Yaskawa INFORM job: DEMO_ROOF_SIDE_0625_3PAINT_18.JBI

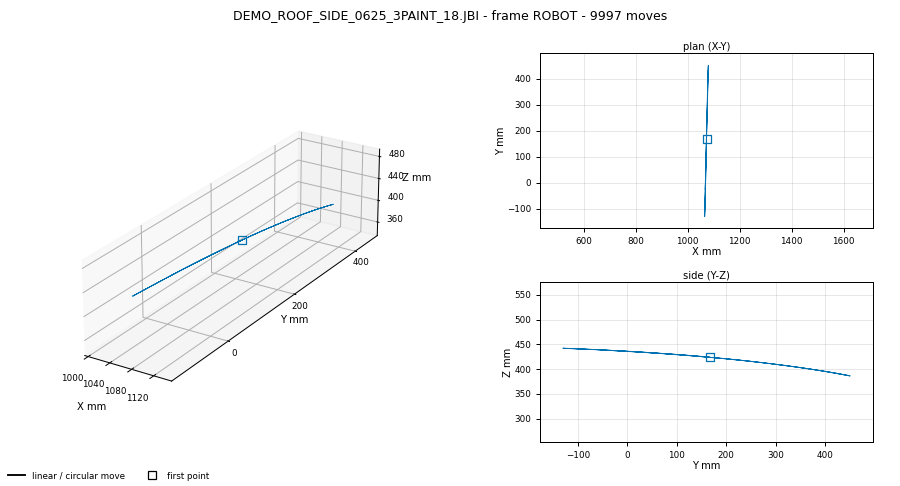
[picture p0: tool path of DEMO_ROOF_SIDE_0625_3PAINT_18.JBI in frame ROBOT, 9997 of 9997 moves have a stored position in this frame; points joined in program order, loops and branches not executed]
/JOB
//NAME DEMO_ROOF_SIDE_0625_3PAINT18
//POS
///NPOS 9997,0,0,0,0,0
///TOOL 0
///USER 0
///POSTYPE ROBOT
///RECTAN
///RCONF 1,0,0,0,0,0,0,0,0,0,0,0,0,0,0,0,0,0,0,0,0,0,0,0
C00000=1073.553,166.231,424.191,173.717,26.118,154.637
C00001=1073.548,165.982,424.213,173.714,26.115,154.636
C00002=1073.541,165.733,424.236,173.713,26.113,154.636
C00003=1073.536,165.484,424.258,173.710,26.110,154.636
C00004=1073.531,165.235,424.280,173.709,26.108,154.635
C00005=1073.525,164.986,424.301,173.707,26.105,154.635
C00006=1073.520,164.737,424.323,173.705,26.102,154.635
C00007=1073.514,164.488,424.345,173.703,26.099,154.634
C00008=1073.509,164.239,424.367,173.701,26.097,154.634
C00009=1073.503,163.990,424.389,173.699,26.094,154.634
C00010=1073.498,163.742,424.411,173.697,26.092,154.633
C00011=1073.492,163.492,424.433,173.695,26.088,154.633
C00012=1073.487,163.244,424.454,173.694,26.086,154.633
C00013=1073.481,162.994,424.477,173.691,26.083,154.632
C00014=1073.476,162.746,424.498,173.690,26.081,154.632
C00015=1073.470,162.496,424.520,173.688,26.078,154.632
C00016=1073.465,162.248,424.541,173.685,26.075,154.631
C00017=1073.459,161.998,424.564,173.684,26.072,154.631
C00018=1073.454,161.750,424.585,173.681,26.069,154.631
C00019=1073.448,161.500,424.607,173.680,26.067,154.630
C00020=1073.443,161.252,424.628,173.678,26.064,154.630
C00021=1073.437,161.002,424.650,173.676,26.061,154.630
C00022=1073.432,160.754,424.672,173.674,26.059,154.629
C00023=1073.426,160.504,424.694,173.672,26.056,154.629
C00024=1073.420,160.255,424.715,173.670,26.054,154.629
C00025=1073.414,160.007,424.736,173.669,26.051,154.628
C00026=1073.409,159.757,424.759,173.666,26.048,154.628
C00027=1073.402,159.475,424.782,173.665,26.045,154.628
C00028=1073.396,159.194,424.807,173.662,26.042,154.627
C00029=1073.390,158.911,424.831,173.660,26.040,154.627
C00030=1073.383,158.630,424.856,173.658,26.036,154.627
C00031=1073.377,158.381,424.877,173.656,26.034,154.626
C00032=1073.372,158.132,424.898,173.654,26.031,154.626
C00033=1073.366,157.882,424.920,173.653,26.028,154.625
C00034=1073.360,157.634,424.941,173.650,26.026,154.625
C00035=1073.355,157.384,424.963,173.649,26.023,154.625
C00036=1073.349,157.136,424.984,173.646,26.020,154.625
C00037=1073.343,156.887,425.006,173.645,26.018,154.624
C00038=1073.338,156.638,425.027,173.643,26.015,154.624
C00039=1073.332,156.388,425.048,173.641,26.013,154.624
C00040=1073.326,156.140,425.070,173.639,26.010,154.623
C00041=1073.321,155.890,425.092,173.637,26.007,154.623
C00042=1073.315,155.641,425.112,173.635,26.005,154.623
C00043=1073.310,155.393,425.134,173.634,26.002,154.622
C00044=1073.304,155.144,425.155,173.631,25.999,154.622
C00045=1073.298,154.895,425.176,173.630,25.997,154.622
C00046=1073.292,154.645,425.197,173.627,25.994,154.621
C00047=1073.287,154.397,425.219,173.626,25.992,154.621
C00048=1073.281,154.147,425.240,173.624,25.989,154.621
C00049=1073.275,153.899,425.262,173.622,25.986,154.620
C00050=1073.269,153.649,425.282,173.621,25.984,154.620
C00051=1073.264,153.401,425.304,173.618,25.981,154.620
C00052=1073.258,153.151,425.326,173.617,25.978,154.619
C00053=1073.253,152.902,425.347,173.614,25.975,154.619
C00054=1073.247,152.654,425.368,173.613,25.973,154.619
C00055=1073.241,152.404,425.389,173.611,25.970,154.618
C00056=1073.236,152.155,425.410,173.609,25.968,154.618
C00057=1073.230,151.906,425.432,173.607,25.965,154.618
C00058=1073.225,151.657,425.452,173.605,25.962,154.617
C00059=1073.219,151.408,425.473,173.604,25.960,154.617
C00060=1073.213,151.159,425.494,173.602,25.957,154.617
C00061=1073.208,150.910,425.516,173.600,25.955,154.616
C00062=1073.201,150.661,425.537,173.598,25.952,154.616
C00063=1073.196,150.412,425.558,173.596,25.949,154.616
C00064=1073.191,150.163,425.579,173.594,25.947,154.615
C00065=1073.185,149.913,425.600,173.593,25.944,154.615
C00066=1073.179,149.665,425.621,173.590,25.941,154.615
C00067=1073.174,149.416,425.642,173.589,25.939,154.615
C00068=1073.168,149.167,425.663,173.587,25.936,154.614
C00069=1073.162,148.917,425.684,173.585,25.933,154.614
C00070=1073.156,148.668,425.706,173.584,25.931,154.613
C00071=1073.150,148.419,425.726,173.581,25.928,154.613
C00072=1073.145,148.171,425.747,173.580,25.925,154.613
C00073=1073.139,147.921,425.768,173.577,25.923,154.613
C00074=1073.133,147.673,425.789,173.576,25.920,154.612
C00075=1073.128,147.423,425.810,173.575,25.918,154.612
C00076=1073.122,147.174,425.831,173.572,25.915,154.612
C00077=1073.117,146.925,425.852,173.571,25.913,154.611
C00078=1073.111,146.676,425.872,173.568,25.909,154.611
C00079=1073.104,146.427,425.893,173.567,25.907,154.611
C00080=1073.099,146.178,425.914,173.565,25.905,154.610
C00081=1073.094,145.929,425.935,173.563,25.902,154.610
C00082=1073.088,145.680,425.956,173.562,25.900,154.610
C00083=1073.082,145.431,425.976,173.559,25.896,154.609
C00084=1073.076,145.182,425.997,173.558,25.894,154.609
C00085=1073.070,144.932,426.018,173.555,25.891,154.609
C00086=1073.065,144.683,426.039,173.554,25.889,154.608
C00087=1073.060,144.435,426.060,173.553,25.886,154.608
C00088=1073.053,144.185,426.080,173.550,25.883,154.608
C00089=1073.048,143.936,426.101,173.549,25.881,154.607
C00090=1073.042,143.687,426.122,173.546,25.878,154.607
C00091=1073.036,143.405,426.145,173.545,25.876,154.607
C00092=1073.029,143.123,426.169,173.543,25.872,154.606
C00093=1073.023,142.841,426.193,173.540,25.869,154.606
C00094=1073.017,142.559,426.215,173.539,25.866,154.606
C00095=1073.011,142.310,426.237,173.537,25.864,154.605
C00096=1073.005,142.060,426.258,173.535,25.861,154.605
C00097=1072.999,141.812,426.278,173.533,25.858,154.605
C00098=1072.994,141.562,426.298,173.532,25.856,154.604
C00099=1072.989,141.313,426.319,173.530,25.853,154.604
C00100=1072.983,141.064,426.340,173.528,25.850,154.604
C00101=1072.977,140.815,426.360,173.526,25.848,154.603
C00102=1072.971,140.566,426.381,173.525,25.845,154.603
C00103=1072.966,140.317,426.401,173.523,25.842,154.603
C00104=1072.959,140.068,426.422,173.521,25.840,154.602
C00105=1072.954,139.818,426.442,173.519,25.837,154.602
C00106=1072.949,139.570,426.463,173.517,25.835,154.602
C00107=1072.943,139.321,426.483,173.516,25.832,154.601
C00108=1072.937,139.071,426.504,173.514,25.829,154.601
C00109=1072.931,138.822,426.524,173.512,25.827,154.601
C00110=1072.926,138.573,426.545,173.511,25.824,154.600
C00111=1072.920,138.324,426.565,173.508,25.822,154.600
C00112=1072.914,138.075,426.585,173.507,25.819,154.600
C00113=1072.908,137.826,426.606,173.505,25.816,154.599
C00114=1072.902,137.577,426.626,173.503,25.814,154.599
C00115=1072.897,137.328,426.647,173.502,25.811,154.599
C00116=1072.891,137.079,426.667,173.499,25.808,154.598
C00117=1072.886,136.830,426.687,173.498,25.806,154.598
C00118=1072.880,136.580,426.708,173.497,25.803,154.598
C00119=1072.874,136.332,426.729,173.494,25.801,154.597
C00120=1072.869,136.083,426.749,173.493,25.798,154.597
C00121=1072.863,135.834,426.769,173.491,25.796,154.597
C00122=1072.858,135.584,426.789,173.489,25.792,154.596
C00123=1072.851,135.334,426.810,173.488,25.790,154.596
C00124=1072.846,135.085,426.830,173.485,25.788,154.596
C00125=1072.840,134.837,426.850,173.484,25.785,154.595
C00126=1072.834,134.587,426.871,173.482,25.782,154.595
C00127=1072.828,134.339,426.891,173.480,25.779,154.595
C00128=1072.823,134.089,426.911,173.479,25.777,154.594
C00129=1072.817,133.841,426.931,173.477,25.774,154.594
C00130=1072.811,133.591,426.952,173.475,25.772,154.594
C00131=1072.805,133.342,426.972,173.473,25.769,154.593
C00132=1072.800,133.093,426.993,173.472,25.766,154.593
C00133=1072.794,132.844,427.013,173.470,25.764,154.593
C00134=1072.789,132.595,427.033,173.468,25.761,154.592
C00135=1072.783,132.346,427.052,173.467,25.759,154.592
C00136=1072.778,132.096,427.073,173.465,25.755,154.592
C00137=1072.772,131.848,427.093,173.463,25.753,154.591
C00138=1072.765,131.598,427.113,173.462,25.750,154.591
C00139=1072.760,131.349,427.134,173.459,25.748,154.591
C00140=1072.754,131.100,427.154,173.458,25.745,154.591
C00141=1072.748,130.851,427.173,173.456,25.743,154.590
C00142=1072.742,130.602,427.193,173.454,25.740,154.590
C00143=1072.737,130.353,427.213,173.453,25.738,154.590
C00144=1072.731,130.103,427.234,173.451,25.735,154.589
C00145=1072.725,129.854,427.254,173.449,25.732,154.589
C00146=1072.719,129.605,427.273,173.447,25.730,154.589
C00147=1072.714,129.356,427.294,173.446,25.727,154.588
C00148=1072.708,129.107,427.313,173.444,25.725,154.588
C00149=1072.702,128.858,427.333,173.442,25.722,154.588
C00150=1072.696,128.609,427.353,173.441,25.719,154.587
C00151=1072.691,128.360,427.373,173.438,25.717,154.587
C00152=1072.684,128.110,427.394,173.437,25.714,154.587
C00153=1072.678,127.861,427.413,173.436,25.712,154.586
C00154=1072.672,127.612,427.433,173.434,25.709,154.586
C00155=1072.666,127.330,427.455,173.432,25.706,154.586
C00156=1072.660,127.047,427.478,173.430,25.703,154.585
C00157=1072.653,126.765,427.500,173.428,25.700,154.585
C00158=1072.647,126.483,427.523,173.426,25.697,154.584
C00159=1072.641,126.234,427.543,173.425,25.695,154.584
C00160=1072.635,125.985,427.562,173.422,25.692,154.584
C00161=1072.630,125.736,427.583,173.421,25.689,154.584
C00162=1072.624,125.487,427.603,173.419,25.687,154.583
C00163=1072.618,125.237,427.622,173.418,25.684,154.583
C00164=1072.612,124.989,427.642,173.416,25.682,154.583
C00165=1072.606,124.739,427.661,173.414,25.679,154.582
C00166=1072.600,124.490,427.681,173.413,25.676,154.582
C00167=1072.595,124.241,427.702,173.410,25.674,154.582
C00168=1072.589,123.992,427.721,173.409,25.671,154.581
C00169=1072.583,123.743,427.741,173.408,25.669,154.581
C00170=1072.578,123.494,427.760,173.405,25.665,154.581
C00171=1072.572,123.245,427.780,173.404,25.663,154.580
C00172=1072.566,122.995,427.799,173.403,25.660,154.580
C00173=1072.561,122.746,427.820,173.401,25.658,154.580
C00174=1072.555,122.497,427.839,173.399,25.655,154.579
C00175=1072.549,122.248,427.859,173.397,25.653,154.579
C00176=1072.543,121.998,427.878,173.396,25.650,154.578
C00177=1072.537,121.750,427.898,173.394,25.647,154.578
C00178=1072.532,121.500,427.917,173.392,25.644,154.578
C00179=1072.526,121.251,427.938,173.391,25.642,154.578
C00180=1072.521,121.002,427.957,173.389,25.640,154.577
C00181=1072.515,120.753,427.977,173.387,25.637,154.577
C00182=1072.509,120.503,427.996,173.386,25.634,154.577
C00183=1072.503,120.254,428.016,173.384,25.631,154.576
C00184=1072.497,120.005,428.036,173.383,25.629,154.576
C00185=1072.492,119.756,428.055,173.381,25.626,154.576
C00186=1072.486,119.507,428.075,173.379,25.624,154.575
C00187=1072.481,119.257,428.095,173.378,25.621,154.575
C00188=1072.475,119.008,428.114,173.375,25.618,154.575
C00189=1072.469,118.759,428.134,173.374,25.615,154.574
C00190=1072.464,118.510,428.153,173.373,25.612,154.574
C00191=1072.458,118.261,428.173,173.371,25.610,154.573
C00192=1072.452,118.012,428.192,173.369,25.607,154.573
C00193=1072.447,117.763,428.211,173.368,25.605,154.573
C00194=1072.441,117.514,428.231,173.366,25.602,154.572
C00195=1072.435,117.264,428.250,173.365,25.600,154.572
C00196=1072.430,117.015,428.270,173.362,25.596,154.572
C00197=1072.424,116.765,428.289,173.361,25.594,154.571
C00198=1072.419,116.517,428.309,173.360,25.591,154.571
C00199=1072.413,116.268,428.328,173.358,25.589,154.571
C00200=1072.408,116.018,428.348,173.356,25.586,154.570
C00201=1072.402,115.769,428.367,173.355,25.583,154.570
C00202=1072.396,115.520,428.387,173.353,25.581,154.570
C00203=1072.390,115.270,428.406,173.352,25.578,154.569
C00204=1072.385,115.022,428.425,173.349,25.575,154.569
C00205=1072.379,114.773,428.445,173.348,25.572,154.569
C00206=1072.373,114.523,428.464,173.347,25.570,154.568
C00207=1072.368,114.274,428.483,173.345,25.567,154.568
C00208=1072.362,114.025,428.503,173.343,25.564,154.568
C00209=1072.356,113.775,428.522,173.342,25.562,154.567
C00210=1072.350,113.526,428.542,173.340,25.559,154.567
C00211=1072.345,113.278,428.561,173.339,25.556,154.567
C00212=1072.340,113.028,428.580,173.336,25.554,154.566
C00213=1072.334,112.779,428.599,173.335,25.551,154.566
C00214=1072.328,112.530,428.618,173.334,25.549,154.566
C00215=1072.322,112.280,428.637,173.332,25.546,154.565
C00216=1072.316,112.031,428.656,173.330,25.543,154.565
C00217=1072.310,111.782,428.676,173.329,25.540,154.565
C00218=1072.305,111.533,428.695,173.327,25.538,154.564
C00219=1072.298,111.251,428.716,173.325,25.535,154.564
C00220=1072.292,110.968,428.738,173.324,25.532,154.563
C00221=1072.285,110.686,428.760,173.321,25.529,154.563
C00222=1072.278,110.403,428.781,173.320,25.526,154.563
C00223=1072.273,110.155,428.800,173.318,25.523,154.562
C00224=1072.267,109.905,428.819,173.316,25.520,154.562
C00225=1072.262,109.656,428.839,173.315,25.518,154.562
C00226=1072.255,109.407,428.857,173.314,25.515,154.561
C00227=1072.249,109.157,428.876,173.312,25.513,154.561
C00228=1072.244,108.908,428.896,173.310,25.510,154.561
C00229=1072.239,108.659,428.915,173.308,25.507,154.560
C00230=1072.232,108.410,428.933,173.307,25.505,154.560
C00231=1072.227,108.160,428.953,173.306,25.502,154.560
C00232=1072.221,107.911,428.972,173.303,25.500,154.559
C00233=1072.214,107.662,428.990,173.302,25.497,154.559
C00234=1072.209,107.413,429.009,173.300,25.495,154.559
C00235=1072.204,107.164,429.029,173.299,25.492,154.558
C00236=1072.197,106.915,429.047,173.298,25.489,154.558
C00237=1072.192,106.665,429.066,173.295,25.486,154.558
C00238=1072.186,106.416,429.086,173.294,25.484,154.557
C00239=1072.181,106.167,429.105,173.293,25.481,154.557
C00240=1072.174,105.918,429.123,173.291,25.479,154.557
C00241=1072.169,105.669,429.142,173.289,25.476,154.556
C00242=1072.163,105.419,429.162,173.288,25.473,154.556
C00243=1072.157,105.171,429.180,173.286,25.470,154.556
C00244=1072.152,104.921,429.198,173.285,25.468,154.555
C00245=1072.146,104.671,429.218,173.283,25.465,154.555
C00246=1072.140,104.423,429.236,173.281,25.463,154.555
C00247=1072.135,104.173,429.255,173.280,25.460,154.554
C00248=1072.129,103.924,429.274,173.278,25.457,154.554
C00249=1072.122,103.675,429.293,173.277,25.455,154.554
C00250=1072.117,103.426,429.312,173.276,25.452,154.553
C00251=1072.112,103.176,429.331,173.273,25.449,154.553
C00252=1072.106,102.927,429.349,173.272,25.446,154.553
C00253=1072.100,102.678,429.368,173.271,25.444,154.552
C00254=1072.094,102.429,429.387,173.269,25.441,154.552
C00255=1072.088,102.180,429.406,173.268,25.439,154.552
C00256=1072.084,101.930,429.424,173.266,25.435,154.551
C00257=1072.077,101.681,429.443,173.264,25.433,154.551
C00258=1072.071,101.432,429.462,173.263,25.430,154.550
C00259=1072.066,101.183,429.481,173.261,25.427,154.550
C00260=1072.060,100.933,429.499,173.260,25.425,154.550
C00261=1072.055,100.684,429.518,173.258,25.422,154.550
C00262=1072.048,100.435,429.537,173.256,25.420,154.549
C00263=1072.042,100.186,429.555,173.255,25.417,154.549
C00264=1072.037,99.936,429.574,173.254,25.414,154.548
C00265=1072.030,99.687,429.592,173.252,25.412,154.548
C00266=1072.025,99.438,429.611,173.250,25.409,154.548
C00267=1072.019,99.189,429.629,173.248,25.407,154.547
C00268=1072.014,98.939,429.648,173.247,25.404,154.547
C00269=1072.007,98.690,429.667,173.246,25.401,154.547
C00270=1072.002,98.441,429.684,173.244,25.399,154.546
C00271=1071.996,98.192,429.704,173.242,25.396,154.546
C00272=1071.990,97.942,429.722,173.241,25.393,154.546
C00273=1071.985,97.693,429.740,173.239,25.391,154.545
C00274=1071.978,97.444,429.759,173.238,25.388,154.545
C00275=1071.973,97.194,429.778,173.236,25.386,154.545
C00276=1071.967,96.945,429.796,173.234,25.382,154.544
C00277=1071.961,96.696,429.815,173.233,25.380,154.544
C00278=1071.956,96.447,429.833,173.231,25.377,154.544
C00279=1071.949,96.198,429.851,173.230,25.375,154.543
C00280=1071.944,95.948,429.870,173.229,25.372,154.543
C00281=1071.938,95.699,429.888,173.227,25.370,154.543
C00282=1071.932,95.450,429.906,173.225,25.367,154.542
C00283=1071.926,95.168,429.927,173.224,25.364,154.542
C00284=1071.919,94.885,429.949,173.221,25.360,154.542
C00285=1071.913,94.604,429.969,173.220,25.358,154.541
C00286=1071.906,94.321,429.990,173.219,25.355,154.541
C00287=1071.900,94.072,430.008,173.217,25.352,154.540
C00288=1071.895,93.822,430.027,173.215,25.349,154.540
C00289=1071.889,93.573,430.045,173.214,25.346,154.540
C00290=1071.883,93.324,430.064,173.212,25.344,154.539
C00291=1071.877,93.074,430.082,173.211,25.341,154.539
C00292=1071.871,92.826,430.100,173.209,25.338,154.539
C00293=1071.866,92.576,430.119,173.207,25.336,154.538
C00294=1071.861,92.327,430.136,173.206,25.333,154.538
C00295=1071.854,92.078,430.155,173.205,25.330,154.538
C00296=1071.849,91.828,430.173,173.203,25.328,154.537
C00297=1071.843,91.579,430.192,173.202,25.325,154.537
C00298=1071.837,91.329,430.210,173.200,25.322,154.537
C00299=1071.832,91.081,430.228,173.198,25.320,154.536
C00300=1071.826,90.831,430.246,173.197,25.317,154.536
C00301=1071.820,90.582,430.264,173.196,25.315,154.536
C00302=1071.814,90.333,430.283,173.194,25.312,154.535
C00303=1071.808,90.084,430.300,173.193,25.309,154.535
C00304=1071.803,89.834,430.319,173.191,25.306,154.535
C00305=1071.796,89.585,430.337,173.189,25.304,154.534
C00306=1071.791,89.335,430.355,173.188,25.301,154.534
C00307=1071.785,89.086,430.373,173.186,25.299,154.534
C00308=1071.779,88.837,430.391,173.185,25.296,154.533
C00309=1071.773,88.588,430.409,173.184,25.293,154.533
C00310=1071.767,88.339,430.427,173.181,25.290,154.532
C00311=1071.762,88.089,430.446,173.180,25.288,154.532
C00312=1071.756,87.840,430.463,173.179,25.285,154.532
C00313=1071.750,87.590,430.481,173.177,25.283,154.532
C00314=1071.744,87.341,430.499,173.176,25.280,154.531
C00315=1071.738,87.092,430.518,173.175,25.277,154.531
C00316=1071.732,86.842,430.536,173.173,25.275,154.530
C00317=1071.726,86.593,430.553,173.171,25.272,154.530
C00318=1071.720,86.344,430.571,173.170,25.269,154.530
C00319=1071.714,86.095,430.589,173.168,25.267,154.529
C00320=1071.708,85.845,430.607,173.167,25.264,154.529
C00321=1071.704,85.596,430.625,173.165,25.262,154.529
C00322=1071.697,85.346,430.643,173.164,25.259,154.528
C00323=1071.692,85.098,430.662,173.162,25.256,154.528
C00324=1071.685,84.848,430.680,173.160,25.253,154.528
C00325=1071.680,84.599,430.697,173.159,25.250,154.527
C00326=1071.674,84.349,430.715,173.158,25.248,154.527
C00327=1071.668,84.100,430.733,173.156,25.245,154.527
C00328=1071.663,83.851,430.750,173.155,25.243,154.526
C00329=1071.656,83.602,430.769,173.154,25.240,154.526
C00330=1071.651,83.353,430.786,173.151,25.237,154.526
C00331=1071.645,83.103,430.804,173.150,25.234,154.525
C00332=1071.639,82.854,430.822,173.149,25.232,154.525
C00333=1071.633,82.605,430.840,173.147,25.229,154.525
C00334=1071.628,82.356,430.857,173.146,25.226,154.524
C00335=1071.622,82.106,430.876,173.145,25.224,154.524
C00336=1071.617,81.857,430.894,173.143,25.221,154.523
C00337=1071.611,81.608,430.911,173.141,25.218,154.523
C00338=1071.605,81.358,430.930,173.140,25.216,154.523
C00339=1071.599,81.109,430.947,173.138,25.213,154.523
C00340=1071.593,80.860,430.965,173.137,25.210,154.522
C00341=1071.588,80.611,430.983,173.136,25.207,154.522
C00342=1071.582,80.362,431.000,173.134,25.205,154.521
C00343=1071.576,80.112,431.018,173.133,25.202,154.521
C00344=1071.570,79.863,431.036,173.131,25.200,154.521
C00345=1071.564,79.613,431.054,173.129,25.197,154.520
C00346=1071.559,79.364,431.071,173.128,25.194,154.520
C00347=1071.552,79.082,431.091,173.127,25.191,154.520
C00348=1071.546,78.800,431.111,173.124,25.188,154.519
C00349=1071.539,78.518,431.131,173.123,25.185,154.519
C00350=1071.532,78.235,431.152,173.122,25.182,154.518
C00351=1071.526,77.986,431.169,173.119,25.179,154.518
C00352=1071.521,77.737,431.186,173.118,25.176,154.518
C00353=1071.515,77.487,431.204,173.117,25.174,154.517
C00354=1071.509,77.237,431.221,173.115,25.171,154.517
C00355=1071.503,76.988,431.239,173.114,25.168,154.517
C00356=1071.498,76.739,431.257,173.113,25.166,154.516
C00357=1071.492,76.490,431.274,173.111,25.163,154.516
C00358=1071.485,76.240,431.292,173.110,25.161,154.516
C00359=1071.480,75.991,431.309,173.108,25.158,154.515
C00360=1071.474,75.742,431.327,173.106,25.155,154.515
C00361=1071.468,75.492,431.345,173.105,25.152,154.515
C00362=1071.463,75.243,431.362,173.104,25.150,154.514
C00363=1071.456,74.994,431.379,173.102,25.147,154.514
C00364=1071.451,74.744,431.396,173.101,25.145,154.514
C00365=1071.445,74.495,431.414,173.100,25.142,154.513
C00366=1071.439,74.246,431.432,173.098,25.140,154.513
C00367=1071.433,73.996,431.449,173.096,25.136,154.513
C00368=1071.427,73.748,431.466,173.095,25.133,154.512
C00369=1071.421,73.497,431.484,173.093,25.131,154.512
C00370=1071.416,73.248,431.501,173.092,25.128,154.511
C00371=1071.410,72.999,431.519,173.091,25.126,154.511
C00372=1071.404,72.750,431.537,173.089,25.123,154.511
C00373=1071.398,72.501,431.554,173.088,25.121,154.511
C00374=1071.393,72.251,431.570,173.087,25.118,154.510
C00375=1071.387,72.001,431.588,173.085,25.115,154.510
C00376=1071.381,71.752,431.606,173.083,25.112,154.509
C00377=1071.375,71.504,431.623,173.082,25.109,154.509
C00378=1071.370,71.254,431.640,173.080,25.107,154.509
C00379=1071.364,71.004,431.658,173.079,25.104,154.508
C00380=1071.357,70.756,431.675,173.077,25.102,154.508
C00381=1071.352,70.507,431.692,173.076,25.099,154.508
C00382=1071.346,70.256,431.709,173.075,25.096,154.507
C00383=1071.340,70.007,431.727,173.074,25.094,154.507
C00384=1071.334,69.758,431.744,173.071,25.090,154.507
C00385=1071.329,69.509,431.761,173.070,25.088,154.506
C00386=1071.323,69.259,431.779,173.069,25.085,154.506
C00387=1071.317,69.010,431.796,173.067,25.083,154.506
C00388=1071.311,68.761,431.813,173.066,25.080,154.505
C00389=1071.305,68.511,431.830,173.064,25.078,154.505
C00390=1071.299,68.262,431.848,173.063,25.075,154.505
C00391=1071.294,68.012,431.864,173.062,25.072,154.504
C00392=1071.288,67.764,431.881,173.060,25.070,154.504
C00393=1071.282,67.513,431.899,173.058,25.066,154.503
C00394=1071.276,67.264,431.916,173.057,25.064,154.503
C00395=1071.270,67.016,431.933,173.056,25.061,154.503
C00396=1071.265,66.766,431.950,173.054,25.059,154.503
C00397=1071.258,66.516,431.967,173.053,25.056,154.502
C00398=1071.253,66.267,431.984,173.051,25.054,154.502
C00399=1071.246,66.018,432.001,173.050,25.051,154.501
C00400=1071.241,65.768,432.018,173.049,25.048,154.501
C00401=1071.235,65.519,432.036,173.047,25.045,154.501
C00402=1071.229,65.270,432.053,173.046,25.043,154.500
C00403=1071.224,65.020,432.070,173.044,25.040,154.500
C00404=1071.217,64.772,432.087,173.043,25.037,154.500
C00405=1071.212,64.521,432.104,173.041,25.035,154.499
C00406=1071.205,64.273,432.121,173.040,25.032,154.499
C00407=1071.200,64.023,432.138,173.038,25.029,154.499
C00408=1071.194,63.774,432.155,173.037,25.027,154.498
C00409=1071.187,63.524,432.171,173.036,25.024,154.498
C00410=1071.182,63.275,432.189,173.034,25.022,154.498
C00411=1071.175,62.992,432.207,173.032,25.019,154.497
C00412=1071.168,62.710,432.227,173.031,25.016,154.497
C00413=1071.161,62.428,432.245,173.030,25.013,154.497
C00414=1071.155,62.145,432.265,173.027,25.010,154.496
C00415=1071.149,61.896,432.281,173.026,25.007,154.496
C00416=1071.142,61.647,432.299,173.025,25.004,154.496
C00417=1071.137,61.397,432.315,173.023,25.002,154.495
C00418=1071.130,61.148,432.332,173.022,24.999,154.495
C00419=1071.125,60.899,432.349,173.021,24.997,154.495
C00420=1071.119,60.649,432.366,173.019,24.994,154.494
C00421=1071.112,60.400,432.383,173.017,24.991,154.494
C00422=1071.107,60.151,432.399,173.016,24.988,154.493
C00423=1071.101,59.901,432.416,173.014,24.986,154.493
C00424=1071.095,59.652,432.433,173.013,24.983,154.493
C00425=1071.089,59.403,432.449,173.012,24.981,154.493
C00426=1071.083,59.153,432.466,173.010,24.978,154.492
C00427=1071.077,58.904,432.483,173.009,24.975,154.492
C00428=1071.071,58.654,432.500,173.008,24.973,154.491
C00429=1071.065,58.405,432.516,173.006,24.970,154.491
C00430=1071.060,58.156,432.534,173.005,24.967,154.491
C00431=1071.054,57.907,432.550,173.003,24.965,154.490
C00432=1071.047,57.657,432.566,173.001,24.962,154.490
C00433=1071.042,57.408,432.584,173.000,24.959,154.490
C00434=1071.036,57.158,432.600,172.999,24.957,154.489
C00435=1071.030,56.909,432.616,172.997,24.954,154.489
C00436=1071.024,56.659,432.633,172.996,24.951,154.489
C00437=1071.018,56.410,432.650,172.995,24.949,154.488
C00438=1071.012,56.161,432.667,172.993,24.946,154.488
C00439=1071.006,55.911,432.683,172.992,24.944,154.488
C00440=1071.000,55.662,432.699,172.991,24.941,154.487
C00441=1070.995,55.412,432.716,172.989,24.938,154.487
C00442=1070.988,55.163,432.733,172.988,24.936,154.487
C00443=1070.982,54.914,432.750,172.986,24.933,154.486
C00444=1070.976,54.665,432.766,172.984,24.930,154.486
C00445=1070.971,54.415,432.783,172.983,24.927,154.486
C00446=1070.965,54.166,432.799,172.982,24.925,154.485
C00447=1070.959,53.917,432.816,172.980,24.922,154.485
C00448=1070.952,53.667,432.832,172.979,24.919,154.485
C00449=1070.947,53.417,432.849,172.978,24.917,154.484
C00450=1070.941,53.168,432.866,172.976,24.914,154.484
C00451=1070.935,52.918,432.882,172.975,24.911,154.484
C00452=1070.929,52.669,432.898,172.974,24.909,154.483
C00453=1070.924,52.419,432.915,172.972,24.906,154.483
C00454=1070.918,52.171,432.932,172.971,24.904,154.483
C00455=1070.912,51.921,432.948,172.969,24.900,154.482
C00456=1070.906,51.672,432.964,172.967,24.898,154.482
C00457=1070.901,51.422,432.981,172.966,24.895,154.482
C00458=1070.895,51.173,432.998,172.965,24.892,154.481
C00459=1070.889,50.924,433.014,172.963,24.890,154.481
C00460=1070.883,50.674,433.030,172.962,24.887,154.480
C00461=1070.877,50.425,433.046,172.961,24.885,154.480
C00462=1070.872,50.175,433.063,172.959,24.882,154.480
C00463=1070.866,49.926,433.079,172.958,24.879,154.479
C00464=1070.860,49.677,433.096,172.957,24.877,154.479
C00465=1070.854,49.427,433.112,172.955,24.874,154.479
C00466=1070.848,49.178,433.128,172.954,24.871,154.478
C00467=1070.843,48.928,433.145,172.953,24.868,154.478
C00468=1070.837,48.679,433.161,172.950,24.866,154.478
C00469=1070.831,48.430,433.178,172.949,24.863,154.477
C00470=1070.825,48.180,433.194,172.948,24.860,154.477
C00471=1070.819,47.931,433.210,172.947,24.858,154.477
C00472=1070.813,47.682,433.226,172.945,24.855,154.476
C00473=1070.808,47.432,433.243,172.944,24.852,154.476
C00474=1070.802,47.183,433.259,172.943,24.849,154.476
C00475=1070.795,46.900,433.278,172.941,24.846,154.475
C00476=1070.789,46.617,433.297,172.939,24.843,154.475
C00477=1070.782,46.335,433.315,172.938,24.840,154.474
C00478=1070.775,46.053,433.333,172.937,24.837,154.474
C00479=1070.769,45.803,433.349,172.935,24.834,154.474
C00480=1070.764,45.554,433.366,172.933,24.832,154.473
C00481=1070.759,45.304,433.382,172.932,24.829,154.473
C00482=1070.753,45.054,433.398,172.931,24.826,154.473
C00483=1070.747,44.805,433.414,172.929,24.824,154.472
C00484=1070.741,44.556,433.431,172.928,24.821,154.472
C00485=1070.735,44.306,433.447,172.926,24.818,154.472
C00486=1070.729,44.057,433.463,172.925,24.815,154.471
C00487=1070.724,43.808,433.480,172.924,24.813,154.471
C00488=1070.719,43.558,433.495,172.923,24.810,154.470
C00489=1070.713,43.309,433.511,172.921,24.807,154.470
C00490=1070.706,43.060,433.527,172.920,24.805,154.470
C00491=1070.700,42.810,433.543,172.919,24.802,154.469
C00492=1070.694,42.561,433.560,172.917,24.800,154.469
C00493=1070.688,42.312,433.576,172.916,24.797,154.469
C00494=1070.682,42.062,433.591,172.914,24.794,154.468
C00495=1070.676,41.812,433.608,172.912,24.791,154.468
C00496=1070.670,41.563,433.624,172.911,24.789,154.468
C00497=1070.665,41.314,433.640,172.910,24.786,154.467
C00498=1070.659,41.064,433.656,172.908,24.784,154.467
C00499=1070.653,40.814,433.672,172.907,24.781,154.467
C00500=1070.647,40.565,433.688,172.906,24.778,154.466
C00501=1070.642,40.316,433.704,172.904,24.775,154.466
C00502=1070.636,40.066,433.720,172.903,24.773,154.466
C00503=1070.630,39.817,433.736,172.902,24.770,154.465
C00504=1070.624,39.568,433.752,172.900,24.768,154.465
C00505=1070.618,39.318,433.767,172.899,24.765,154.465
C00506=1070.612,39.069,433.783,172.898,24.762,154.464
C00507=1070.606,38.819,433.800,172.896,24.760,154.464
C00508=1070.600,38.570,433.816,172.894,24.757,154.464
C00509=1070.595,38.321,433.831,172.893,24.754,154.463
C00510=1070.589,38.071,433.847,172.891,24.752,154.463
C00511=1070.583,37.822,433.864,172.890,24.749,154.463
C00512=1070.577,37.572,433.879,172.889,24.746,154.462
C00513=1070.571,37.323,433.895,172.888,24.743,154.462
C00514=1070.565,37.073,433.910,172.886,24.741,154.462
C00515=1070.559,36.824,433.927,172.885,24.738,154.461
C00516=1070.553,36.574,433.943,172.883,24.736,154.461
C00517=1070.547,36.325,433.958,172.882,24.733,154.461
C00518=1070.541,36.076,433.974,172.881,24.730,154.460
C00519=1070.536,35.826,433.989,172.879,24.728,154.460
C00520=1070.529,35.577,434.005,172.878,24.725,154.460
C00521=1070.523,35.328,434.021,172.877,24.723,154.459
C00522=1070.517,35.078,434.037,172.876,24.720,154.459
C00523=1070.511,34.828,434.053,172.873,24.717,154.459
C00524=1070.505,34.579,434.068,172.872,24.714,154.458
C00525=1070.500,34.330,434.084,172.871,24.712,154.458
C00526=1070.494,34.080,434.099,172.869,24.710,154.458
C00527=1070.487,33.831,434.115,172.868,24.707,154.457
C00528=1070.482,33.581,434.130,172.867,24.704,154.457
C00529=1070.476,33.332,434.147,172.865,24.701,154.457
C00530=1070.470,33.082,434.162,172.864,24.699,154.456
C00531=1070.464,32.833,434.178,172.863,24.696,154.456
C00532=1070.458,32.583,434.193,172.861,24.694,154.456
C00533=1070.452,32.334,434.209,172.860,24.691,154.455
C00534=1070.446,32.084,434.224,172.859,24.688,154.455
C00535=1070.440,31.835,434.241,172.857,24.686,154.455
C00536=1070.435,31.586,434.256,172.856,24.683,154.454
C00537=1070.428,31.337,434.271,172.855,24.680,154.454
C00538=1070.423,31.087,434.287,172.853,24.678,154.454
C00539=1070.416,30.804,434.305,172.851,24.675,154.453
C00540=1070.410,30.522,434.323,172.850,24.672,154.453
C00541=1070.402,30.239,434.340,172.849,24.669,154.452
C00542=1070.396,29.957,434.357,172.846,24.666,154.452
C00543=1070.390,29.707,434.373,172.845,24.663,154.452
C00544=1070.385,29.457,434.389,172.844,24.660,154.451
C00545=1070.378,29.208,434.404,172.842,24.658,154.451
C00546=1070.373,28.959,434.420,172.841,24.655,154.451
C00547=1070.367,28.709,434.435,172.840,24.653,154.450
C00548=1070.361,28.460,434.451,172.838,24.650,154.450
C00549=1070.354,28.210,434.466,172.837,24.647,154.450
C00550=1070.349,27.960,434.481,172.836,24.645,154.449
C00551=1070.343,27.712,434.497,172.835,24.642,154.449
C00552=1070.337,27.462,434.512,172.833,24.640,154.449
C00553=1070.331,27.212,434.528,172.832,24.637,154.449
C00554=1070.325,26.963,434.543,172.831,24.634,154.448
C00555=1070.319,26.714,434.558,172.828,24.632,154.448
C00556=1070.313,26.464,434.573,172.827,24.629,154.447
C00557=1070.307,26.215,434.590,172.826,24.626,154.447
C00558=1070.301,25.965,434.605,172.824,24.624,154.447
C00559=1070.296,25.716,434.620,172.823,24.621,154.447
C00560=1070.289,25.466,434.635,172.822,24.619,154.446
C00561=1070.283,25.217,434.651,172.820,24.616,154.446
C00562=1070.277,24.967,434.666,172.819,24.613,154.446
C00563=1070.271,24.718,434.681,172.818,24.611,154.445
C00564=1070.266,24.468,434.696,172.816,24.608,154.445
C00565=1070.259,24.219,434.711,172.815,24.606,154.445
C00566=1070.254,23.970,434.727,172.814,24.603,154.444
C00567=1070.247,23.720,434.742,172.812,24.601,154.444
C00568=1070.242,23.470,434.757,172.811,24.598,154.444
C00569=1070.235,23.221,434.772,172.810,24.595,154.443
C00570=1070.230,22.971,434.788,172.808,24.593,154.443
C00571=1070.224,22.722,434.803,172.807,24.590,154.443
C00572=1070.217,22.473,434.818,172.805,24.587,154.442
C00573=1070.212,22.223,434.833,172.803,24.585,154.442
C00574=1070.206,21.974,434.848,172.802,24.582,154.442
C00575=1070.200,21.724,434.864,172.801,24.580,154.441
C00576=1070.194,21.475,434.878,172.799,24.577,154.441
C00577=1070.188,21.225,434.895,172.798,24.574,154.441
C00578=1070.182,20.976,434.910,172.797,24.572,154.440
C00579=1070.176,20.727,434.924,172.795,24.569,154.440
C00580=1070.171,20.477,434.940,172.794,24.567,154.440
C00581=1070.164,20.227,434.955,172.793,24.564,154.439
C00582=1070.159,19.978,434.970,172.791,24.561,154.439
C00583=1070.153,19.728,434.985,172.790,24.559,154.439
C00584=1070.146,19.479,435.000,172.789,24.557,154.438
C00585=1070.141,19.229,435.015,172.787,24.554,154.438
C00586=1070.135,18.980,435.030,172.786,24.551,154.438
C00587=1070.129,18.730,435.045,172.785,24.549,154.438
C00588=1070.123,18.481,435.059,172.783,24.546,154.437
C00589=1070.117,18.231,435.075,172.782,24.544,154.437
C00590=1070.111,17.982,435.089,172.780,24.541,154.437
C00591=1070.105,17.733,435.104,172.779,24.538,154.436
C00592=1070.099,17.483,435.120,172.777,24.536,154.436
C00593=1070.094,17.234,435.135,172.776,24.533,154.436
C00594=1070.087,16.984,435.149,172.775,24.530,154.435
C00595=1070.081,16.734,435.164,172.773,24.528,154.435
C00596=1070.076,16.485,435.180,172.772,24.525,154.435
C00597=1070.069,16.235,435.195,172.771,24.523,154.434
C00598=1070.064,15.986,435.209,172.769,24.520,154.434
C00599=1070.058,15.736,435.225,172.768,24.517,154.434
C00600=1070.052,15.487,435.240,172.767,24.515,154.433
C00601=1070.046,15.238,435.254,172.765,24.513,154.433
C00602=1070.039,14.988,435.269,172.764,24.510,154.433
C00603=1070.033,14.707,435.286,172.763,24.507,154.432
C00604=1070.027,14.426,435.303,172.760,24.504,154.432
C00605=1070.020,14.144,435.320,172.759,24.501,154.432
C00606=1070.013,13.863,435.336,172.758,24.499,154.431
C00607=1070.006,13.614,435.351,172.757,24.496,154.431
C00608=1070.001,13.364,435.366,172.754,24.493,154.431
C00609=1069.995,13.115,435.381,172.753,24.491,154.430
C00610=1069.989,12.865,435.396,172.751,24.488,154.430
C00611=1069.983,12.616,435.410,172.750,24.485,154.430
C00612=1069.976,12.367,435.425,172.749,24.483,154.429
C00613=1069.971,12.117,435.439,172.747,24.481,154.429
C00614=1069.965,11.867,435.454,172.746,24.478,154.429
C00615=1069.958,11.618,435.469,172.745,24.475,154.429
C00616=1069.952,11.369,435.484,172.743,24.473,154.428
C00617=1069.946,11.119,435.499,172.742,24.470,154.428
C00618=1069.940,10.870,435.513,172.741,24.468,154.428
C00619=1069.934,10.620,435.527,172.739,24.466,154.427
C00620=1069.928,10.371,435.542,172.738,24.463,154.427
C00621=1069.922,10.121,435.557,172.737,24.460,154.427
C00622=1069.916,9.872,435.572,172.735,24.458,154.426
C00623=1069.910,9.622,435.586,172.734,24.456,154.426
C00624=1069.904,9.372,435.601,172.733,24.453,154.426
C00625=1069.898,9.123,435.615,172.731,24.450,154.425
C00626=1069.892,8.874,435.630,172.729,24.448,154.425
C00627=1069.886,8.624,435.644,172.728,24.445,154.425
C00628=1069.880,8.374,435.660,172.726,24.442,154.425
C00629=1069.875,8.125,435.674,172.725,24.440,154.424
C00630=1069.868,7.876,435.689,172.724,24.438,154.424
C00631=1069.863,7.626,435.703,172.722,24.435,154.424
C00632=1069.856,7.376,435.718,172.721,24.433,154.423
C00633=1069.851,7.127,435.732,172.720,24.430,154.423
C00634=1069.845,6.877,435.747,172.718,24.428,154.423
C00635=1069.839,6.628,435.761,172.717,24.425,154.423
C00636=1069.832,6.378,435.776,172.716,24.423,154.422
C00637=1069.827,6.129,435.790,172.714,24.420,154.422
C00638=1069.821,5.879,435.805,172.713,24.417,154.422
C00639=1069.815,5.630,435.820,172.712,24.415,154.421
C00640=1069.809,5.380,435.834,172.710,24.413,154.421
C00641=1069.803,5.131,435.848,172.709,24.410,154.421
C00642=1069.797,4.881,435.863,172.708,24.407,154.420
C00643=1069.791,4.632,435.877,172.706,24.405,154.420
C00644=1069.784,4.382,435.892,172.705,24.403,154.420
C00645=1069.778,4.133,435.905,172.703,24.400,154.420
C00646=1069.773,3.884,435.920,172.701,24.397,154.419
C00647=1069.767,3.634,435.934,172.700,24.395,154.419
C00648=1069.761,3.385,435.949,172.699,24.392,154.419
C00649=1069.754,3.135,435.964,172.697,24.390,154.418
C00650=1069.749,2.885,435.978,172.696,24.387,154.418
C00651=1069.743,2.636,435.993,172.695,24.384,154.418
C00652=1069.737,2.386,436.006,172.693,24.382,154.417
C00653=1069.731,2.137,436.021,172.692,24.380,154.417
C00654=1069.725,1.887,436.035,172.691,24.377,154.417
C00655=1069.719,1.638,436.050,172.689,24.374,154.416
C00656=1069.713,1.388,436.064,172.688,24.372,154.416
C00657=1069.708,1.139,436.079,172.687,24.370,154.416
C00658=1069.702,0.889,436.093,172.685,24.367,154.416
C00659=1069.696,0.640,436.107,172.684,24.364,154.415
C00660=1069.690,0.390,436.121,172.683,24.362,154.415
C00661=1069.684,0.140,436.136,172.681,24.360,154.415
C00662=1069.678,-0.109,436.150,172.680,24.357,154.414
C00663=1069.673,-0.358,436.165,172.678,24.354,154.414
C00664=1069.666,-0.608,436.178,172.676,24.351,154.414
C00665=1069.660,-0.858,436.192,172.675,24.349,154.413
C00666=1069.655,-1.107,436.207,172.674,24.347,154.413
C00667=1069.648,-1.386,436.223,172.672,24.344,154.413
C00668=1069.642,-1.666,436.239,172.671,24.341,154.412
C00669=1069.635,-1.945,436.255,172.669,24.338,154.412
C00670=1069.628,-2.224,436.271,172.668,24.336,154.412
C00671=1069.622,-2.474,436.285,172.666,24.333,154.411
C00672=1069.617,-2.723,436.299,172.665,24.330,154.411
C00673=1069.610,-2.973,436.314,172.664,24.328,154.411
C00674=1069.605,-3.223,436.327,172.662,24.326,154.411
C00675=1069.599,-3.472,436.341,172.661,24.323,154.410
C00676=1069.592,-3.721,436.356,172.660,24.321,154.410
C00677=1069.587,-3.971,436.370,172.658,24.318,154.410
C00678=1069.581,-4.220,436.384,172.657,24.315,154.409
C00679=1069.574,-4.470,436.398,172.656,24.313,154.409
C00680=1069.569,-4.719,436.412,172.654,24.311,154.409
C00681=1069.563,-4.970,436.426,172.653,24.308,154.409
C00682=1069.556,-5.218,436.440,172.651,24.306,154.408
C00683=1069.551,-5.468,436.454,172.649,24.303,154.408
C00684=1069.544,-5.718,436.468,172.648,24.301,154.408
C00685=1069.538,-5.967,436.482,172.646,24.298,154.407
C00686=1069.532,-6.216,436.496,172.645,24.296,154.407
C00687=1069.526,-6.467,436.510,172.644,24.294,154.407
C00688=1069.520,-6.716,436.523,172.642,24.291,154.407
C00689=1069.514,-6.965,436.538,172.641,24.289,154.406
C00690=1069.508,-7.215,436.551,172.640,24.286,154.406
C00691=1069.502,-7.465,436.565,172.638,24.284,154.406
C00692=1069.497,-7.714,436.579,172.637,24.282,154.406
C00693=1069.490,-7.963,436.594,172.636,24.279,154.405
C00694=1069.484,-8.213,436.607,172.634,24.277,154.405
C00695=1069.479,-8.463,436.621,172.633,24.275,154.405
C00696=1069.472,-8.713,436.635,172.631,24.272,154.404
C00697=1069.466,-8.962,436.649,172.630,24.270,154.404
C00698=1069.460,-9.211,436.663,172.629,24.267,154.404
C00699=1069.454,-9.460,436.677,172.626,24.265,154.404
C00700=1069.448,-9.711,436.691,172.625,24.262,154.403
C00701=1069.442,-9.960,436.704,172.624,24.259,154.403
C00702=1069.437,-10.209,436.718,172.622,24.257,154.403
C00703=1069.430,-10.459,436.731,172.621,24.255,154.402
C00704=1069.424,-10.709,436.745,172.620,24.252,154.402
C00705=1069.418,-10.958,436.760,172.618,24.250,154.402
C00706=1069.412,-11.207,436.773,172.617,24.247,154.402
C00707=1069.407,-11.457,436.787,172.616,24.245,154.401
C00708=1069.400,-11.707,436.801,172.614,24.243,154.401
C00709=1069.394,-11.956,436.815,172.613,24.240,154.401
C00710=1069.389,-12.206,436.829,172.612,24.238,154.401
C00711=1069.383,-12.455,436.842,172.610,24.235,154.400
C00712=1069.377,-12.705,436.856,172.609,24.233,154.400
C00713=1069.370,-12.955,436.869,172.608,24.231,154.400
C00714=1069.365,-13.204,436.883,172.606,24.228,154.399
C00715=1069.359,-13.454,436.896,172.605,24.226,154.399
C00716=1069.353,-13.704,436.911,172.603,24.223,154.399
C00717=1069.346,-13.953,436.924,172.601,24.221,154.399
C00718=1069.341,-14.203,436.938,172.600,24.218,154.398
C00719=1069.336,-14.452,436.952,172.598,24.216,154.398
C00720=1069.329,-14.702,436.965,172.597,24.214,154.398
C00721=1069.323,-14.952,436.979,172.596,24.211,154.398
C00722=1069.317,-15.201,436.992,172.594,24.209,154.397
C00723=1069.311,-15.450,437.006,172.593,24.206,154.397
C00724=1069.305,-15.700,437.020,172.592,24.204,154.397
C00725=1069.299,-15.949,437.033,172.590,24.202,154.397
C00726=1069.293,-16.199,437.047,172.589,24.200,154.396
C00727=1069.287,-16.449,437.060,172.587,24.197,154.396
C00728=1069.281,-16.698,437.074,172.586,24.195,154.396
C00729=1069.275,-16.948,437.088,172.585,24.193,154.395
C00730=1069.268,-17.198,437.101,172.583,24.190,154.395
C00731=1069.262,-17.475,437.117,172.581,24.187,154.395
C00732=1069.255,-17.753,437.131,172.580,24.185,154.395
C00733=1069.248,-18.030,437.146,172.578,24.182,154.394
C00734=1069.242,-18.308,437.160,172.577,24.180,154.394
C00735=1069.236,-18.557,437.174,172.575,24.177,154.394
C00736=1069.230,-18.807,437.188,172.573,24.175,154.394
C00737=1069.223,-19.057,437.201,172.572,24.173,154.393
C00738=1069.218,-19.306,437.215,172.571,24.170,154.393
C00739=1069.211,-19.555,437.228,172.569,24.168,154.393
C00740=1069.205,-19.805,437.242,172.568,24.166,154.393
C00741=1069.200,-20.054,437.255,172.567,24.163,154.392
C00742=1069.194,-20.304,437.268,172.565,24.161,154.392
C00743=1069.187,-20.554,437.282,172.564,24.159,154.392
C00744=1069.181,-20.804,437.296,172.562,24.156,154.392
C00745=1069.175,-21.053,437.309,172.561,24.154,154.391
C00746=1069.169,-21.302,437.322,172.560,24.152,154.391
C00747=1069.164,-21.552,437.335,172.558,24.149,154.391
C00748=1069.158,-21.802,437.348,172.557,24.147,154.390
C00749=1069.151,-22.051,437.362,172.556,24.144,154.390
C00750=1069.145,-22.301,437.376,172.554,24.143,154.390
C00751=1069.139,-22.550,437.389,172.553,24.140,154.390
C00752=1069.133,-22.800,437.402,172.550,24.138,154.390
C00753=1069.127,-23.050,437.415,172.549,24.135,154.389
C00754=1069.122,-23.299,437.429,172.548,24.133,154.389
C00755=1069.115,-23.548,437.442,172.546,24.130,154.389
C00756=1069.109,-23.798,437.455,172.545,24.128,154.389
C00757=1069.104,-24.048,437.469,172.543,24.126,154.388
C00758=1069.098,-24.297,437.482,172.542,24.124,154.388
C00759=1069.092,-24.547,437.494,172.541,24.121,154.388
C00760=1069.086,-24.796,437.508,172.539,24.119,154.387
C00761=1069.080,-25.046,437.522,172.538,24.116,154.387
C00762=1069.073,-25.296,437.535,172.537,24.115,154.387
C00763=1069.067,-25.546,437.548,172.535,24.112,154.387
C00764=1069.061,-25.795,437.561,172.534,24.110,154.387
C00765=1069.056,-26.045,437.575,172.532,24.107,154.386
C00766=1069.050,-26.294,437.587,172.531,24.105,154.386
C00767=1069.044,-26.544,437.601,172.530,24.103,154.386
C00768=1069.038,-26.794,437.613,172.527,24.100,154.386
C00769=1069.032,-27.043,437.627,172.526,24.098,154.385
C00770=1069.026,-27.292,437.640,172.525,24.096,154.385
C00771=1069.020,-27.542,437.653,172.523,24.094,154.385
C00772=1069.014,-27.792,437.666,172.522,24.091,154.385
C00773=1069.008,-28.041,437.679,172.520,24.089,154.384
C00774=1069.002,-28.291,437.692,172.519,24.087,154.384
C00775=1068.996,-28.540,437.705,172.518,24.085,154.384
C00776=1068.990,-28.790,437.718,172.516,24.082,154.384
C00777=1068.983,-29.039,437.731,172.515,24.080,154.383
C00778=1068.977,-29.290,437.744,172.513,24.078,154.383
C00779=1068.971,-29.539,437.757,172.512,24.076,154.383
C00780=1068.964,-29.788,437.771,172.511,24.073,154.383
C00781=1068.959,-30.038,437.783,172.509,24.072,154.383
C00782=1068.952,-30.287,437.796,172.508,24.069,154.382
C00783=1068.946,-30.537,437.809,172.506,24.067,154.382
C00784=1068.940,-30.787,437.822,172.504,24.065,154.382
C00785=1068.934,-31.036,437.835,172.503,24.062,154.382
C00786=1068.928,-31.286,437.848,172.501,24.060,154.381
C00787=1068.922,-31.536,437.861,172.500,24.058,154.381
C00788=1068.916,-31.785,437.874,172.498,24.055,154.381
C00789=1068.911,-32.035,437.887,172.497,24.054,154.381
C00790=1068.905,-32.284,437.900,172.496,24.051,154.380
C00791=1068.899,-32.534,437.913,172.494,24.049,154.380
C00792=1068.892,-32.783,437.926,172.493,24.047,154.380
C00793=1068.887,-33.033,437.939,172.491,24.045,154.380
C00794=1068.881,-33.283,437.951,172.490,24.042,154.380
C00795=1068.874,-33.560,437.966,172.489,24.040,154.379
C00796=1068.867,-33.836,437.979,172.486,24.037,154.379
C00797=1068.860,-34.113,437.994,172.485,24.035,154.379
C00798=1068.853,-34.390,438.008,172.484,24.033,154.379
C00799=1068.847,-34.640,438.021,172.482,24.030,154.378
C00800=1068.841,-34.890,438.033,172.481,24.028,154.378
C00801=1068.835,-35.139,438.047,172.479,24.026,154.378
C00802=1068.829,-35.389,438.059,172.477,24.023,154.378
C00803=1068.823,-35.639,438.072,172.476,24.022,154.378
C00804=1068.818,-35.887,438.085,172.474,24.019,154.377
C00805=1068.812,-36.137,438.097,172.473,24.017,154.377
C00806=1068.806,-36.387,438.110,172.471,24.015,154.377
C00807=1068.800,-36.636,438.123,172.470,24.012,154.377
C00808=1068.794,-36.886,438.136,172.469,24.011,154.376
C00809=1068.788,-37.136,438.148,172.467,24.008,154.376
C00810=1068.782,-37.385,438.161,172.466,24.006,154.376
C00811=1068.776,-37.635,438.174,172.464,24.004,154.376
C00812=1068.770,-37.885,438.187,172.463,24.002,154.375
C00813=1068.764,-38.134,438.200,172.462,24.000,154.375
C00814=1068.758,-38.383,438.212,172.460,23.997,154.375
C00815=1068.752,-38.633,438.225,172.459,23.995,154.375
C00816=1068.746,-38.883,438.238,172.457,23.993,154.375
C00817=1068.740,-39.132,438.250,172.456,23.991,154.374
C00818=1068.734,-39.382,438.262,172.454,23.988,154.374
C00819=1068.728,-39.632,438.275,172.452,23.987,154.374
C00820=1068.721,-39.881,438.288,172.451,23.984,154.374
C00821=1068.716,-40.131,438.301,172.449,23.982,154.374
C00822=1068.709,-40.381,438.313,172.448,23.980,154.373
C00823=1068.703,-40.630,438.325,172.446,23.978,154.373
C00824=1068.697,-40.880,438.338,172.445,23.976,154.373
C00825=1068.691,-41.130,438.351,172.444,23.974,154.373
C00826=1068.685,-41.378,438.363,172.442,23.971,154.373
C00827=1068.679,-41.628,438.375,172.441,23.970,154.372
C00828=1068.673,-41.878,438.388,172.439,23.968,154.372
C00829=1068.667,-42.128,438.400,172.438,23.965,154.372
C00830=1068.660,-42.377,438.413,172.436,23.963,154.372
C00831=1068.654,-42.627,438.426,172.435,23.961,154.372
C00832=1068.648,-42.877,438.438,172.433,23.959,154.371
C00833=1068.642,-43.127,438.451,172.432,23.957,154.371
C00834=1068.636,-43.376,438.462,172.430,23.955,154.371
C00835=1068.630,-43.625,438.475,172.428,23.953,154.371
C00836=1068.625,-43.875,438.487,172.427,23.950,154.371
C00837=1068.618,-44.125,438.499,172.425,23.949,154.371
C00838=1068.612,-44.374,438.513,172.424,23.946,154.370
C00839=1068.606,-44.624,438.525,172.423,23.944,154.370
C00840=1068.601,-44.873,438.537,172.421,23.942,154.370
C00841=1068.594,-45.123,438.549,172.420,23.940,154.370
C00842=1068.588,-45.373,438.562,172.418,23.938,154.370
C00843=1068.582,-45.623,438.574,172.417,23.936,154.369
C00844=1068.575,-45.872,438.586,172.415,23.934,154.369
C00845=1068.569,-46.122,438.599,172.414,23.932,154.369
C00846=1068.564,-46.371,438.611,172.413,23.930,154.369
C00847=1068.558,-46.621,438.624,172.411,23.928,154.369
C00848=1068.552,-46.871,438.636,172.410,23.925,154.368
C00849=1068.546,-47.121,438.648,172.408,23.924,154.368
C00850=1068.540,-47.370,438.661,172.406,23.921,154.368
C00851=1068.534,-47.619,438.672,172.404,23.919,154.368
C00852=1068.528,-47.869,438.685,172.403,23.917,154.368
C00853=1068.522,-48.119,438.697,172.401,23.915,154.367
C00854=1068.515,-48.369,438.709,172.400,23.913,154.367
C00855=1068.510,-48.618,438.722,172.399,23.911,154.367
C00856=1068.504,-48.868,438.734,172.397,23.909,154.367
C00857=1068.497,-49.117,438.746,172.396,23.907,154.367
C00858=1068.492,-49.367,438.759,172.394,23.905,154.366
C00859=1068.485,-49.644,438.772,172.393,23.902,154.366
C00860=1068.478,-49.921,438.786,172.391,23.900,154.366
C00861=1068.472,-50.199,438.799,172.389,23.898,154.366
C00862=1068.465,-50.476,438.813,172.388,23.896,154.366
C00863=1068.459,-50.726,438.825,172.386,23.894,154.365
C00864=1068.453,-50.975,438.836,172.385,23.892,154.365
C00865=1068.447,-51.225,438.849,172.383,23.890,154.365
C00866=1068.440,-51.474,438.861,172.382,23.888,154.365
C00867=1068.434,-51.724,438.874,172.380,23.886,154.365
C00868=1068.428,-51.974,438.885,172.378,23.884,154.365
C00869=1068.422,-52.223,438.896,172.376,23.882,154.365
C00870=1068.416,-52.473,438.909,172.375,23.880,154.364
C00871=1068.409,-52.723,438.921,172.374,23.878,154.364
C00872=1068.403,-52.972,438.933,172.372,23.876,154.364
C00873=1068.397,-53.222,438.945,172.371,23.874,154.364
C00874=1068.391,-53.471,438.957,172.369,23.872,154.364
C00875=1068.385,-53.721,438.969,172.368,23.870,154.364
C00876=1068.378,-53.971,438.981,172.366,23.869,154.363
C00877=1068.372,-54.221,438.993,172.365,23.867,154.363
C00878=1068.366,-54.470,439.005,172.363,23.865,154.363
C00879=1068.360,-54.719,439.017,172.362,23.862,154.363
C00880=1068.354,-54.970,439.029,172.360,23.861,154.363
C00881=1068.347,-55.219,439.041,172.359,23.859,154.363
C00882=1068.341,-55.468,439.052,172.357,23.857,154.362
C00883=1068.335,-55.718,439.065,172.356,23.855,154.362
C00884=1068.329,-55.968,439.076,172.354,23.853,154.362
C00885=1068.323,-56.217,439.088,172.352,23.851,154.362
C00886=1068.317,-56.467,439.100,172.350,23.849,154.362
C00887=1068.311,-56.717,439.112,172.349,23.847,154.362
C00888=1068.304,-56.967,439.123,172.347,23.845,154.362
C00889=1068.299,-57.216,439.136,172.346,23.844,154.361
C00890=1068.292,-57.466,439.148,172.344,23.842,154.361
C00891=1068.286,-57.716,439.159,172.343,23.839,154.361
C00892=1068.281,-57.965,439.171,172.342,23.837,154.361
C00893=1068.274,-58.214,439.183,172.340,23.836,154.361
C00894=1068.267,-58.464,439.195,172.339,23.834,154.361
C00895=1068.262,-58.714,439.206,172.337,23.832,154.360
C00896=1068.256,-58.963,439.218,172.336,23.830,154.360
C00897=1068.249,-59.213,439.230,172.334,23.828,154.360
C00898=1068.243,-59.462,439.241,172.333,23.826,154.360
C00899=1068.237,-59.712,439.254,172.331,23.824,154.360
C00900=1068.231,-59.963,439.265,172.330,23.823,154.360
C00901=1068.225,-60.211,439.277,172.328,23.821,154.360
C00902=1068.219,-60.461,439.289,172.326,23.819,154.360
C00903=1068.213,-60.712,439.300,172.324,23.817,154.359
C00904=1068.207,-60.960,439.312,172.323,23.815,154.359
C00905=1068.201,-61.211,439.324,172.321,23.813,154.359
C00906=1068.194,-61.460,439.336,172.320,23.811,154.359
C00907=1068.188,-61.709,439.347,172.318,23.809,154.359
C00908=1068.182,-61.960,439.359,172.317,23.807,154.359
C00909=1068.177,-62.209,439.371,172.315,23.806,154.358
C00910=1068.170,-62.459,439.382,172.314,23.804,154.358
C00911=1068.164,-62.708,439.394,172.312,23.802,154.358
C00912=1068.158,-62.958,439.405,172.311,23.800,154.358
C00913=1068.152,-63.208,439.417,172.309,23.798,154.358
C00914=1068.146,-63.457,439.429,172.308,23.796,154.358
C00915=1068.140,-63.707,439.440,172.306,23.794,154.358
C00916=1068.134,-63.956,439.452,172.305,23.793,154.357
C00917=1068.128,-64.206,439.464,172.303,23.791,154.357
C00918=1068.121,-64.456,439.476,172.302,23.789,154.357
C00919=1068.116,-64.705,439.487,172.300,23.787,154.357
C00920=1068.110,-64.955,439.499,172.298,23.785,154.357
C00921=1068.104,-65.205,439.510,172.296,23.784,154.357
C00922=1068.097,-65.454,439.522,172.295,23.782,154.357
C00923=1068.091,-65.733,439.535,172.293,23.779,154.357
C00924=1068.084,-66.011,439.548,172.292,23.777,154.356
C00925=1068.077,-66.290,439.560,172.290,23.776,154.356
C00926=1068.071,-66.569,439.573,172.288,23.773,154.356
C00927=1068.065,-66.818,439.585,172.287,23.771,154.356
C00928=1068.059,-67.068,439.596,172.285,23.770,154.356
C00929=1068.053,-67.317,439.607,172.284,23.768,154.356
C00930=1068.046,-67.567,439.619,172.282,23.766,154.356
C00931=1068.041,-67.817,439.631,172.280,23.765,154.356
C00932=1068.035,-68.067,439.642,172.279,23.763,154.355
C00933=1068.029,-68.316,439.653,172.277,23.761,154.355
C00934=1068.022,-68.566,439.665,172.276,23.759,154.355
C00935=1068.017,-68.815,439.676,172.274,23.757,154.355
C00936=1068.011,-69.066,439.688,172.273,23.755,154.355
C00937=1068.005,-69.315,439.699,172.271,23.753,154.355
C00938=1067.999,-69.565,439.710,172.270,23.752,154.355
C00939=1067.993,-69.814,439.721,172.268,23.750,154.355
C00940=1067.986,-70.064,439.733,172.267,23.748,154.354
C00941=1067.981,-70.314,439.745,172.264,23.746,154.354
C00942=1067.975,-70.564,439.756,172.263,23.744,154.354
C00943=1067.969,-70.813,439.768,172.261,23.743,154.354
C00944=1067.963,-71.063,439.779,172.260,23.741,154.354
C00945=1067.957,-71.312,439.790,172.258,23.739,154.354
C00946=1067.951,-71.562,439.802,172.257,23.737,154.354
C00947=1067.945,-71.812,439.813,172.255,23.736,154.354
C00948=1067.939,-72.061,439.824,172.254,23.734,154.353
C00949=1067.933,-72.311,439.836,172.252,23.732,154.353
C00950=1067.927,-72.560,439.847,172.251,23.730,154.353
C00951=1067.921,-72.810,439.858,172.249,23.729,154.353
C00952=1067.916,-73.060,439.870,172.248,23.727,154.353
C00953=1067.910,-73.309,439.881,172.246,23.725,154.353
C00954=1067.903,-73.559,439.892,172.245,23.723,154.353
C00955=1067.898,-73.809,439.903,172.243,23.721,154.353
C00956=1067.891,-74.059,439.915,172.242,23.720,154.352
C00957=1067.885,-74.309,439.925,172.240,23.718,154.352
C00958=1067.879,-74.557,439.937,172.239,23.716,154.352
C00959=1067.873,-74.808,439.948,172.237,23.715,154.352
C00960=1067.867,-75.057,439.959,172.235,23.713,154.352
C00961=1067.861,-75.307,439.970,172.234,23.711,154.352
C00962=1067.855,-75.557,439.981,172.232,23.710,154.352
C00963=1067.849,-75.807,439.993,172.230,23.708,154.352
C00964=1067.843,-76.056,440.004,172.228,23.706,154.352
C00965=1067.837,-76.305,440.015,172.227,23.705,154.352
C00966=1067.831,-76.556,440.026,172.225,23.703,154.351
C00967=1067.824,-76.805,440.037,172.224,23.701,154.351
C00968=1067.818,-77.055,440.048,172.222,23.700,154.351
C00969=1067.812,-77.304,440.059,172.221,23.698,154.351
C00970=1067.806,-77.555,440.070,172.219,23.696,154.351
C00971=1067.800,-77.803,440.081,172.218,23.695,154.351
C00972=1067.794,-78.053,440.092,172.216,23.693,154.351
C00973=1067.788,-78.303,440.104,172.214,23.691,154.351
C00974=1067.782,-78.553,440.114,172.213,23.690,154.351
C00975=1067.776,-78.802,440.125,172.211,23.688,154.351
C00976=1067.770,-79.052,440.137,172.210,23.686,154.351
C00977=1067.764,-79.302,440.147,172.208,23.685,154.351
C00978=1067.757,-79.552,440.158,172.207,23.683,154.350
C00979=1067.751,-79.801,440.169,172.205,23.682,154.350
C00980=1067.746,-80.051,440.180,172.203,23.680,154.350
C00981=1067.739,-80.301,440.191,172.202,23.679,154.350
C00982=1067.734,-80.550,440.202,172.200,23.677,154.350
C00983=1067.726,-80.800,440.213,172.199,23.676,154.350
C00984=1067.721,-81.050,440.224,172.197,23.674,154.350
C00985=1067.715,-81.299,440.234,172.196,23.673,154.350
C00986=1067.708,-81.549,440.245,172.194,23.671,154.350
C00987=1067.701,-81.829,440.257,172.191,23.669,154.350
C00988=1067.694,-82.110,440.270,172.190,23.667,154.350
C00989=1067.688,-82.391,440.282,172.188,23.666,154.350
C00990=1067.680,-82.672,440.294,172.186,23.664,154.350
C00991=1067.674,-82.922,440.305,172.184,23.662,154.350
C00992=1067.668,-83.171,440.316,172.183,23.661,154.350
C00993=1067.661,-83.421,440.326,172.181,23.659,154.349
C00994=1067.656,-83.670,440.337,172.180,23.658,154.349
C00995=1067.650,-83.920,440.348,172.178,23.656,154.349
C00996=1067.644,-84.170,440.359,172.176,23.655,154.349
C00997=1067.637,-84.420,440.369,172.175,23.653,154.349
C00998=1067.632,-84.669,440.380,172.173,23.652,154.349
C00999=1067.625,-84.920,440.391,172.172,23.650,154.349
C01000=1067.619,-85.169,440.401,172.170,23.649,154.349
C01001=1067.613,-85.418,440.412,172.168,23.647,154.349
C01002=1067.607,-85.668,440.424,172.167,23.646,154.349
C01003=1067.600,-85.918,440.434,172.165,23.645,154.349
C01004=1067.595,-86.167,440.445,172.164,23.643,154.349
C01005=1067.588,-86.418,440.455,172.162,23.641,154.349
C01006=1067.582,-86.667,440.465,172.160,23.640,154.349
C01007=1067.576,-86.917,440.476,172.159,23.638,154.349
C01008=1067.569,-87.166,440.487,172.157,23.637,154.348
C01009=1067.563,-87.416,440.498,172.156,23.636,154.348
C01010=1067.558,-87.665,440.509,172.154,23.634,154.348
C01011=1067.552,-87.915,440.518,172.152,23.632,154.348
C01012=1067.545,-88.165,440.530,172.151,23.631,154.348
C01013=1067.539,-88.415,440.540,172.149,23.630,154.348
C01014=1067.533,-88.664,440.551,172.148,23.628,154.348
C01015=1067.527,-88.914,440.562,172.146,23.627,154.348
C01016=1067.521,-89.164,440.572,172.144,23.625,154.348
C01017=1067.515,-89.414,440.582,172.143,23.624,154.348
C01018=1067.509,-89.663,440.593,172.141,23.622,154.348
C01019=1067.503,-89.912,440.604,172.140,23.621,154.348
C01020=1067.496,-90.163,440.614,172.137,23.619,154.348
C01021=1067.491,-90.413,440.625,172.135,23.618,154.348
C01022=1067.484,-90.662,440.635,172.134,23.616,154.348
C01023=1067.479,-90.911,440.646,172.132,23.615,154.348
C01024=1067.472,-91.162,440.656,172.131,23.614,154.348
C01025=1067.466,-91.411,440.667,172.129,23.612,154.348
C01026=1067.460,-91.661,440.678,172.127,23.611,154.348
C01027=1067.454,-91.910,440.687,172.126,23.609,154.348
C01028=1067.448,-92.160,440.698,172.124,23.608,154.348
C01029=1067.441,-92.410,440.709,172.122,23.606,154.348
C01030=1067.436,-92.660,440.719,172.121,23.605,154.348
C01031=1067.430,-92.909,440.730,172.119,23.604,154.348
C01032=1067.424,-93.159,440.740,172.118,23.602,154.347
C01033=1067.418,-93.409,440.750,172.116,23.601,154.347
C01034=1067.411,-93.659,440.761,172.114,23.599,154.347
C01035=1067.405,-93.908,440.772,172.113,23.598,154.347
C01036=1067.400,-94.158,440.782,172.111,23.597,154.347
C01037=1067.393,-94.407,440.792,172.109,23.596,154.347
C01038=1067.388,-94.658,440.803,172.108,23.594,154.347
C01039=1067.382,-94.907,440.813,172.106,23.592,154.347
C01040=1067.375,-95.157,440.824,172.105,23.591,154.347
C01041=1067.369,-95.407,440.834,172.103,23.590,154.347
C01042=1067.363,-95.656,440.845,172.101,23.588,154.347
C01043=1067.357,-95.906,440.854,172.100,23.587,154.347
C01044=1067.351,-96.155,440.865,172.098,23.586,154.347
C01045=1067.346,-96.405,440.876,172.096,23.585,154.347
C01046=1067.339,-96.655,440.885,172.095,23.583,154.347
C01047=1067.334,-96.904,440.896,172.093,23.581,154.347
C01048=1067.327,-97.155,440.906,172.092,23.580,154.347
C01049=1067.321,-97.404,440.917,172.090,23.579,154.347
C01050=1067.315,-97.654,440.927,172.088,23.577,154.347
C01051=1067.308,-97.937,440.938,172.087,23.576,154.347
C01052=1067.301,-98.220,440.950,172.084,23.575,154.347
C01053=1067.294,-98.502,440.961,172.082,23.573,154.347
C01054=1067.287,-98.785,440.973,172.081,23.572,154.347
C01055=1067.282,-99.035,440.983,172.079,23.571,154.347
C01056=1067.275,-99.286,440.993,172.078,23.569,154.347
C01057=1067.269,-99.535,441.004,172.076,23.568,154.347
C01058=1067.263,-99.785,441.014,172.074,23.567,154.347
C01059=1067.256,-100.034,441.024,172.073,23.565,154.347
C01060=1067.251,-100.284,441.034,172.071,23.564,154.347
C01061=1067.244,-100.534,441.044,172.069,23.563,154.347
C01062=1067.238,-100.783,441.054,172.067,23.562,154.347
C01063=1067.233,-101.033,441.065,172.066,23.561,154.347
C01064=1067.226,-101.283,441.075,172.064,23.560,154.347
C01065=1067.220,-101.533,441.084,172.063,23.558,154.347
C01066=1067.213,-101.782,441.095,172.061,23.557,154.347
C01067=1067.208,-102.033,441.105,172.059,23.556,154.347
C01068=1067.201,-102.282,441.115,172.058,23.554,154.347
C01069=1067.195,-102.531,441.125,172.056,23.553,154.347
C01070=1067.190,-102.782,441.135,172.054,23.552,154.347
C01071=1067.183,-103.031,441.145,172.052,23.551,154.347
C01072=1067.177,-103.281,441.155,172.051,23.550,154.347
C01073=1067.172,-103.531,441.165,172.049,23.548,154.347
C01074=1067.165,-103.780,441.175,172.048,23.547,154.347
C01075=1067.158,-104.030,441.185,172.046,23.546,154.347
C01076=1067.152,-104.280,441.195,172.044,23.545,154.347
C01077=1067.146,-104.530,441.205,172.042,23.544,154.347
C01078=1067.140,-104.779,441.215,172.041,23.542,154.347
C01079=1067.134,-105.029,441.225,172.039,23.541,154.347
C01080=1067.128,-105.279,441.235,172.037,23.540,154.347
C01081=1067.122,-105.529,441.245,172.036,23.539,154.347
C01082=1067.116,-105.778,441.255,172.034,23.538,154.347
C01083=1067.109,-106.028,441.265,172.032,23.537,154.347
C01084=1067.104,-106.278,441.275,172.031,23.535,154.347
C01085=1067.098,-106.527,441.285,172.029,23.534,154.347
C01086=1067.092,-106.777,441.294,172.027,23.533,154.347
C01087=1067.085,-107.026,441.304,172.026,23.532,154.347
C01088=1067.079,-107.276,441.314,172.024,23.531,154.347
C01089=1067.074,-107.526,441.324,172.022,23.530,154.347
C01090=1067.067,-107.776,441.334,172.020,23.529,154.347
C01091=1067.061,-108.025,441.344,172.019,23.527,154.347
C01092=1067.055,-108.275,441.354,172.017,23.527,154.347
C01093=1067.049,-108.525,441.363,172.015,23.525,154.347
C01094=1067.042,-108.775,441.373,172.014,23.524,154.347
C01095=1067.036,-109.024,441.382,172.012,23.523,154.347
C01096=1067.031,-109.274,441.393,172.010,23.522,154.347
C01097=1067.024,-109.524,441.403,172.009,23.521,154.347
C01098=1067.018,-109.774,441.412,172.007,23.520,154.347
C01099=1067.012,-110.023,441.422,172.005,23.519,154.347
C01100=1067.006,-110.273,441.431,172.003,23.518,154.347
C01101=1067.000,-110.523,441.441,172.002,23.517,154.347
C01102=1066.993,-110.772,441.451,172.000,23.515,154.347
C01103=1066.987,-111.022,441.461,171.998,23.515,154.348
C01104=1066.981,-111.272,441.470,171.997,23.513,154.348
C01105=1066.975,-111.522,441.480,171.995,23.512,154.348
C01106=1066.969,-111.772,441.490,171.993,23.511,154.348
C01107=1066.963,-112.021,441.500,171.991,23.510,154.348
C01108=1066.957,-112.271,441.509,171.990,23.509,154.348
C01109=1066.951,-112.521,441.519,171.988,23.508,154.348
C01110=1066.944,-112.770,441.529,171.986,23.507,154.348
C01111=1066.938,-113.020,441.539,171.985,23.506,154.348
C01112=1066.932,-113.270,441.548,171.983,23.505,154.348
C01113=1066.926,-113.520,441.558,171.981,23.504,154.348
C01114=1066.920,-113.769,441.567,171.979,23.503,154.348
C01115=1066.913,-114.051,441.578,171.978,23.502,154.348
C01116=1066.906,-114.331,441.589,171.976,23.501,154.348
C01117=1066.899,-114.613,441.599,171.973,23.499,154.348
C01118=1066.892,-114.893,441.610,171.971,23.499,154.348
C01119=1066.886,-115.143,441.620,171.970,23.497,154.348
C01120=1066.880,-115.393,441.629,171.968,23.497,154.348
C01121=1066.874,-115.643,441.639,171.966,23.495,154.348
C01122=1066.867,-115.892,441.648,171.965,23.495,154.348
C01123=1066.861,-116.142,441.658,171.963,23.493,154.348
C01124=1066.855,-116.392,441.668,171.961,23.493,154.349
C01125=1066.849,-116.642,441.677,171.959,23.492,154.349
C01126=1066.843,-116.892,441.687,171.958,23.490,154.349
C01127=1066.837,-117.141,441.696,171.956,23.490,154.349
C01128=1066.831,-117.390,441.706,171.954,23.488,154.349
C01129=1066.825,-117.640,441.715,171.952,23.488,154.349
C01130=1066.819,-117.890,441.725,171.951,23.487,154.349
C01131=1066.812,-118.140,441.734,171.949,23.486,154.349
C01132=1066.806,-118.390,441.744,171.947,23.485,154.349
C01133=1066.800,-118.639,441.753,171.946,23.485,154.349
C01134=1066.794,-118.890,441.762,171.945,23.483,154.349
C01135=1066.787,-119.139,441.771,171.943,23.483,154.349
C01136=1066.781,-119.389,441.781,171.941,23.482,154.349
C01137=1066.775,-119.639,441.790,171.939,23.481,154.349
C01138=1066.769,-119.888,441.800,171.937,23.480,154.349
C01139=1066.763,-120.138,441.809,171.936,23.479,154.350
C01140=1066.757,-120.388,441.819,171.934,23.478,154.350
C01141=1066.751,-120.637,441.828,171.932,23.477,154.350
C01142=1066.745,-120.887,441.838,171.930,23.476,154.350
C01143=1066.739,-121.138,441.847,171.929,23.475,154.350
C01144=1066.732,-121.387,441.856,171.927,23.474,154.350
C01145=1066.726,-121.636,441.865,171.925,23.474,154.350
C01146=1066.720,-121.886,441.874,171.923,23.473,154.350
C01147=1066.714,-122.136,441.884,171.922,23.472,154.350
C01148=1066.708,-122.386,441.893,171.920,23.471,154.350
C01149=1066.702,-122.636,441.902,171.918,23.470,154.350
C01150=1066.695,-122.885,441.911,171.916,23.469,154.350
C01151=1066.690,-123.135,441.921,171.914,23.469,154.351
C01152=1066.683,-123.384,441.930,171.913,23.467,154.351
C01153=1066.677,-123.634,441.940,171.911,23.467,154.351
C01154=1066.671,-123.885,441.949,171.909,23.466,154.351
C01155=1066.665,-124.134,441.958,171.907,23.465,154.351
C01156=1066.658,-124.384,441.967,171.905,23.464,154.351
C01157=1066.653,-124.633,441.976,171.904,23.463,154.351
C01158=1066.647,-124.883,441.985,171.902,23.462,154.351
C01159=1066.641,-125.133,441.995,171.901,23.462,154.351
C01160=1066.634,-125.383,442.004,171.899,23.461,154.351
C01161=1066.628,-125.632,442.013,171.897,23.461,154.351
C01162=1066.622,-125.882,442.022,171.896,23.460,154.351
C01163=1066.616,-126.132,442.031,171.894,23.459,154.352
C01164=1066.609,-126.381,442.040,171.892,23.458,154.352
C01165=1066.603,-126.632,442.049,171.890,23.458,154.352
C01166=1066.597,-126.882,442.059,171.888,23.457,154.352
C01167=1066.591,-127.130,442.067,171.887,23.456,154.352
C01168=1066.585,-127.380,442.077,171.885,23.455,154.352
C01169=1066.579,-127.631,442.086,171.883,23.454,154.352
C01170=1066.573,-127.880,442.095,171.881,23.453,154.352
C01171=1066.568,-128.131,442.105,171.880,23.452,154.352
C01172=1066.564,-128.382,442.115,171.878,23.450,154.352
C01173=1066.564,-128.632,442.126,171.877,23.448,154.352
C01174=1066.564,-128.883,442.139,171.876,23.444,154.351
C01175=1066.566,-129.136,442.152,171.875,23.441,154.351
C01176=1066.570,-129.388,442.165,171.875,23.436,154.350
C01177=1066.575,-129.639,442.179,171.875,23.431,154.349
C01178=1066.583,-129.889,442.195,171.874,23.425,154.348
C01179=1066.197,-129.912,442.019,171.827,23.572,154.381
C01180=1066.189,-129.661,442.003,171.828,23.578,154.382
C01181=1066.183,-129.410,441.989,171.827,23.583,154.383
C01182=1066.179,-129.158,441.975,171.828,23.588,154.384
C01183=1066.178,-128.905,441.962,171.829,23.592,154.384
C01184=1066.177,-128.655,441.950,171.830,23.595,154.385
C01185=1066.179,-128.405,441.938,171.831,23.597,154.385
C01186=1066.181,-128.154,441.928,171.832,23.600,154.385
C01187=1066.186,-127.903,441.918,171.834,23.601,154.385
C01188=1066.192,-127.653,441.909,171.836,23.602,154.385
C01189=1066.198,-127.403,441.900,171.838,23.603,154.385
C01190=1066.204,-127.153,441.890,171.840,23.603,154.385
C01191=1066.210,-126.905,441.882,171.841,23.604,154.385
C01192=1066.216,-126.654,441.873,171.843,23.605,154.385
C01193=1066.222,-126.404,441.863,171.845,23.606,154.384
C01194=1066.229,-126.155,441.854,171.847,23.606,154.384
C01195=1066.235,-125.904,441.845,171.849,23.607,154.384
C01196=1066.241,-125.655,441.836,171.849,23.608,154.384
C01197=1066.247,-125.405,441.827,171.851,23.609,154.384
C01198=1066.254,-125.156,441.818,171.853,23.609,154.384
C01199=1066.260,-124.906,441.809,171.855,23.610,154.384
C01200=1066.266,-124.656,441.799,171.857,23.611,154.384
C01201=1066.272,-124.407,441.790,171.858,23.612,154.384
C01202=1066.278,-124.157,441.781,171.860,23.612,154.384
C01203=1066.284,-123.907,441.772,171.862,23.613,154.383
C01204=1066.290,-123.657,441.763,171.864,23.614,154.383
C01205=1066.297,-123.407,441.753,171.866,23.615,154.383
C01206=1066.303,-123.157,441.743,171.867,23.616,154.383
C01207=1066.308,-122.908,441.735,171.869,23.616,154.383
C01208=1066.315,-122.658,441.726,171.871,23.618,154.383
C01209=1066.321,-122.408,441.716,171.873,23.618,154.383
C01210=1066.327,-122.159,441.707,171.874,23.619,154.383
C01211=1066.334,-121.909,441.697,171.876,23.620,154.383
C01212=1066.340,-121.659,441.688,171.878,23.621,154.383
C01213=1066.345,-121.409,441.679,171.880,23.622,154.383
C01214=1066.351,-121.159,441.670,171.882,23.623,154.383
C01215=1066.358,-120.910,441.661,171.883,23.623,154.383
C01216=1066.364,-120.660,441.651,171.885,23.625,154.383
C01217=1066.370,-120.410,441.642,171.887,23.625,154.382
C01218=1066.377,-120.161,441.632,171.889,23.626,154.382
C01219=1066.383,-119.911,441.622,171.890,23.627,154.382
C01220=1066.388,-119.661,441.614,171.892,23.628,154.382
C01221=1066.394,-119.411,441.604,171.894,23.629,154.382
C01222=1066.400,-119.161,441.595,171.896,23.630,154.382
C01223=1066.406,-118.912,441.585,171.897,23.631,154.382
C01224=1066.413,-118.662,441.576,171.899,23.632,154.382
C01225=1066.420,-118.412,441.567,171.901,23.633,154.382
C01226=1066.426,-118.163,441.557,171.902,23.633,154.382
C01227=1066.432,-117.913,441.548,171.904,23.634,154.382
C01228=1066.438,-117.663,441.538,171.905,23.635,154.382
C01229=1066.444,-117.413,441.528,171.907,23.636,154.382
C01230=1066.450,-117.164,441.519,171.909,23.637,154.382
C01231=1066.456,-116.914,441.510,171.911,23.638,154.382
C01232=1066.462,-116.665,441.500,171.912,23.639,154.381
C01233=1066.468,-116.415,441.491,171.914,23.640,154.381
C01234=1066.475,-116.165,441.481,171.916,23.641,154.381
C01235=1066.481,-115.915,441.471,171.918,23.641,154.381
C01236=1066.487,-115.665,441.462,171.919,23.643,154.381
C01237=1066.493,-115.416,441.452,171.921,23.643,154.381
C01238=1066.499,-115.166,441.443,171.923,23.645,154.381
C01239=1066.505,-114.916,441.433,171.925,23.645,154.381
C01240=1066.512,-114.635,441.423,171.926,23.647,154.381
C01241=1066.519,-114.354,441.412,171.929,23.648,154.381
C01242=1066.526,-114.073,441.401,171.931,23.649,154.381
C01243=1066.533,-113.791,441.390,171.932,23.650,154.381
C01244=1066.539,-113.542,441.381,171.934,23.651,154.381
C01245=1066.545,-113.293,441.371,171.936,23.652,154.381
C01246=1066.551,-113.043,441.362,171.938,23.653,154.381
C01247=1066.558,-112.793,441.352,171.939,23.654,154.381
C01248=1066.564,-112.543,441.342,171.941,23.655,154.381
C01249=1066.569,-112.293,441.332,171.943,23.657,154.381
C01250=1066.575,-112.043,441.323,171.945,23.657,154.380
C01251=1066.581,-111.793,441.313,171.946,23.659,154.380
C01252=1066.588,-111.544,441.304,171.948,23.659,154.380
C01253=1066.594,-111.294,441.294,171.950,23.661,154.380
C01254=1066.600,-111.045,441.284,171.951,23.662,154.380
C01255=1066.606,-110.795,441.274,171.953,23.663,154.380
C01256=1066.613,-110.545,441.265,171.955,23.664,154.380
C01257=1066.619,-110.295,441.255,171.957,23.665,154.380
C01258=1066.625,-110.046,441.245,171.958,23.666,154.380
C01259=1066.631,-109.796,441.236,171.960,23.667,154.380
C01260=1066.637,-109.546,441.225,171.962,23.668,154.380
C01261=1066.643,-109.296,441.215,171.963,23.669,154.380
C01262=1066.649,-109.047,441.206,171.965,23.670,154.380
C01263=1066.655,-108.797,441.196,171.967,23.671,154.380
C01264=1066.662,-108.547,441.187,171.969,23.672,154.380
C01265=1066.668,-108.298,441.176,171.970,23.673,154.380
C01266=1066.674,-108.048,441.167,171.972,23.674,154.380
C01267=1066.680,-107.798,441.157,171.974,23.676,154.380
C01268=1066.686,-107.548,441.147,171.975,23.677,154.380
C01269=1066.692,-107.298,441.138,171.977,23.678,154.380
C01270=1066.698,-107.049,441.127,171.979,23.679,154.380
C01271=1066.705,-106.799,441.118,171.980,23.680,154.380
C01272=1066.711,-106.550,441.108,171.982,23.681,154.380
C01273=1066.717,-106.299,441.098,171.984,23.682,154.380
C01274=1066.723,-106.050,441.087,171.986,23.684,154.380
C01275=1066.730,-105.800,441.078,171.987,23.685,154.380
C01276=1066.736,-105.550,441.068,171.989,23.686,154.380
C01277=1066.741,-105.301,441.057,171.991,23.687,154.380
C01278=1066.748,-105.051,441.048,171.992,23.688,154.380
C01279=1066.754,-104.801,441.038,171.994,23.690,154.380
C01280=1066.760,-104.552,441.028,171.996,23.691,154.380
C01281=1066.766,-104.302,441.018,171.997,23.692,154.380
C01282=1066.772,-104.052,441.008,171.999,23.693,154.380
C01283=1066.778,-103.803,440.998,172.001,23.694,154.380
C01284=1066.784,-103.553,440.988,172.002,23.695,154.380
C01285=1066.790,-103.303,440.978,172.004,23.697,154.380
C01286=1066.796,-103.054,440.968,172.006,23.698,154.380
C01287=1066.803,-102.804,440.958,172.008,23.699,154.380
C01288=1066.808,-102.554,440.948,172.009,23.700,154.380
C01289=1066.815,-102.304,440.938,172.011,23.701,154.380
C01290=1066.821,-102.054,440.928,172.012,23.703,154.380
C01291=1066.827,-101.804,440.917,172.014,23.704,154.380
C01292=1066.833,-101.555,440.908,172.016,23.705,154.380
C01293=1066.839,-101.305,440.898,172.017,23.707,154.380
C01294=1066.845,-101.055,440.887,172.019,23.708,154.380
C01295=1066.851,-100.806,440.878,172.021,23.709,154.380
C01296=1066.858,-100.556,440.867,172.023,23.710,154.380
C01297=1066.863,-100.306,440.857,172.024,23.711,154.380
C01298=1066.870,-100.057,440.847,172.026,23.712,154.380
C01299=1066.876,-99.807,440.837,172.028,23.714,154.380
C01300=1066.882,-99.557,440.826,172.029,23.715,154.380
C01301=1066.888,-99.307,440.816,172.031,23.716,154.380
C01302=1066.895,-99.058,440.807,172.033,23.718,154.380
C01303=1066.900,-98.808,440.796,172.034,23.719,154.380
C01304=1066.907,-98.525,440.784,172.036,23.720,154.380
C01305=1066.914,-98.241,440.773,172.038,23.722,154.380
C01306=1066.921,-97.958,440.762,172.040,23.723,154.380
C01307=1066.929,-97.675,440.750,172.042,23.724,154.380
C01308=1066.934,-97.426,440.739,172.043,23.726,154.380
C01309=1066.941,-97.176,440.729,172.045,23.727,154.380
C01310=1066.946,-96.927,440.719,172.047,23.728,154.380
C01311=1066.952,-96.677,440.709,172.048,23.730,154.380
C01312=1066.959,-96.427,440.698,172.050,23.731,154.380
C01313=1066.965,-96.177,440.688,172.051,23.733,154.380
C01314=1066.971,-95.927,440.677,172.053,23.734,154.380
C01315=1066.977,-95.678,440.668,172.055,23.735,154.380
C01316=1066.983,-95.428,440.657,172.056,23.737,154.380
C01317=1066.988,-95.179,440.646,172.058,23.738,154.380
C01318=1066.995,-94.929,440.636,172.060,23.739,154.380
C01319=1067.001,-94.679,440.625,172.061,23.740,154.380
C01320=1067.007,-94.429,440.616,172.063,23.742,154.380
C01321=1067.013,-94.179,440.605,172.065,23.744,154.380
C01322=1067.019,-93.930,440.594,172.067,23.745,154.380
C01323=1067.025,-93.680,440.584,172.069,23.747,154.380
C01324=1067.030,-93.431,440.573,172.070,23.748,154.380
C01325=1067.038,-93.181,440.563,172.072,23.749,154.380
C01326=1067.043,-92.931,440.553,172.074,23.751,154.380
C01327=1067.049,-92.681,440.542,172.075,23.752,154.380
C01328=1067.055,-92.432,440.531,172.077,23.754,154.380
C01329=1067.061,-92.182,440.522,172.079,23.755,154.380
C01330=1067.068,-91.932,440.511,172.080,23.756,154.380
C01331=1067.073,-91.682,440.500,172.082,23.758,154.381
C01332=1067.080,-91.433,440.490,172.083,23.759,154.381
C01333=1067.085,-91.183,440.479,172.085,23.761,154.381
C01334=1067.092,-90.934,440.469,172.087,23.762,154.381
C01335=1067.098,-90.684,440.458,172.088,23.764,154.381
C01336=1067.104,-90.434,440.448,172.090,23.765,154.381
C01337=1067.110,-90.185,440.437,172.091,23.766,154.381
C01338=1067.116,-89.935,440.427,172.093,23.768,154.381
C01339=1067.122,-89.685,440.415,172.095,23.769,154.381
C01340=1067.128,-89.435,440.406,172.096,23.771,154.381
C01341=1067.134,-89.186,440.395,172.098,23.772,154.381
C01342=1067.141,-88.936,440.385,172.100,23.773,154.381
C01343=1067.147,-88.686,440.373,172.101,23.775,154.381
C01344=1067.152,-88.436,440.363,172.103,23.776,154.381
C01345=1067.159,-88.187,440.353,172.104,23.778,154.381
C01346=1067.165,-87.937,440.342,172.106,23.779,154.381
C01347=1067.171,-87.687,440.331,172.108,23.781,154.381
C01348=1067.177,-87.438,440.320,172.109,23.782,154.381
C01349=1067.183,-87.188,440.310,172.111,23.784,154.381
C01350=1067.189,-86.938,440.299,172.112,23.785,154.382
C01351=1067.196,-86.689,440.289,172.114,23.787,154.382
C01352=1067.201,-86.439,440.278,172.116,23.788,154.382
C01353=1067.208,-86.189,440.267,172.117,23.790,154.382
C01354=1067.214,-85.940,440.256,172.119,23.791,154.382
C01355=1067.220,-85.690,440.245,172.120,23.792,154.382
C01356=1067.227,-85.440,440.236,172.122,23.794,154.382
C01357=1067.232,-85.190,440.225,172.124,23.796,154.382
C01358=1067.238,-84.941,440.214,172.126,23.797,154.382
C01359=1067.245,-84.691,440.203,172.128,23.799,154.382
C01360=1067.251,-84.441,440.192,172.129,23.800,154.382
C01361=1067.257,-84.192,440.181,172.131,23.802,154.382
C01362=1067.263,-83.942,440.170,172.132,23.803,154.382
C01363=1067.270,-83.693,440.160,172.134,23.805,154.382
C01364=1067.275,-83.443,440.149,172.136,23.806,154.382
C01365=1067.282,-83.193,440.138,172.137,23.808,154.382
C01366=1067.288,-82.944,440.127,172.139,23.809,154.382
C01367=1067.294,-82.694,440.117,172.140,23.811,154.382
C01368=1067.301,-82.413,440.105,172.142,23.812,154.383
C01369=1067.307,-82.132,440.092,172.144,23.814,154.383
C01370=1067.315,-81.851,440.081,172.146,23.816,154.383
C01371=1067.321,-81.571,440.068,172.148,23.818,154.383
C01372=1067.328,-81.320,440.057,172.149,23.819,154.383
C01373=1067.334,-81.071,440.047,172.151,23.821,154.383
C01374=1067.341,-80.821,440.036,172.152,23.822,154.383
C01375=1067.346,-80.572,440.025,172.154,23.824,154.383
C01376=1067.352,-80.322,440.014,172.156,23.825,154.383
C01377=1067.359,-80.072,440.003,172.157,23.827,154.383
C01378=1067.365,-79.823,439.992,172.159,23.828,154.383
C01379=1067.371,-79.572,439.981,172.160,23.830,154.383
C01380=1067.377,-79.323,439.970,172.162,23.832,154.383
C01381=1067.383,-79.073,439.959,172.163,23.833,154.384
C01382=1067.389,-78.823,439.948,172.165,23.835,154.384
C01383=1067.395,-78.574,439.936,172.167,23.837,154.384
C01384=1067.401,-78.324,439.925,172.169,23.838,154.384
C01385=1067.408,-78.075,439.915,172.171,23.840,154.384
C01386=1067.414,-77.826,439.904,172.172,23.842,154.384
C01387=1067.420,-77.575,439.893,172.174,23.843,154.384
C01388=1067.426,-77.326,439.882,172.175,23.845,154.384
C01389=1067.432,-77.076,439.871,172.177,23.846,154.384
C01390=1067.438,-76.826,439.860,172.178,23.848,154.384
C01391=1067.444,-76.577,439.849,172.180,23.850,154.384
C01392=1067.450,-76.327,439.837,172.182,23.851,154.384
C01393=1067.456,-76.078,439.826,172.183,23.853,154.385
C01394=1067.462,-75.827,439.815,172.185,23.855,154.385
C01395=1067.468,-75.578,439.804,172.186,23.856,154.385
C01396=1067.474,-75.328,439.793,172.188,23.858,154.385
C01397=1067.480,-75.078,439.782,172.189,23.860,154.385
C01398=1067.486,-74.829,439.770,172.191,23.861,154.385
C01399=1067.493,-74.579,439.759,172.192,23.863,154.385
C01400=1067.498,-74.330,439.748,172.194,23.865,154.385
C01401=1067.505,-74.080,439.737,172.196,23.866,154.385
C01402=1067.510,-73.830,439.726,172.197,23.868,154.386
C01403=1067.517,-73.580,439.714,172.199,23.870,154.386
C01404=1067.523,-73.331,439.703,172.200,23.872,154.386
C01405=1067.528,-73.082,439.692,172.202,23.873,154.386
C01406=1067.535,-72.831,439.681,172.203,23.875,154.386
C01407=1067.541,-72.582,439.669,172.206,23.877,154.386
C01408=1067.547,-72.332,439.658,172.207,23.879,154.386
C01409=1067.552,-72.082,439.647,172.209,23.881,154.386
C01410=1067.559,-71.832,439.635,172.210,23.882,154.386
C01411=1067.565,-71.583,439.624,172.212,23.884,154.386
C01412=1067.570,-71.334,439.613,172.213,23.886,154.387
C01413=1067.577,-71.084,439.602,172.215,23.888,154.387
C01414=1067.582,-70.835,439.590,172.216,23.890,154.387
C01415=1067.588,-70.584,439.578,172.218,23.891,154.387
C01416=1067.594,-70.335,439.567,172.219,23.893,154.387
C01417=1067.601,-70.085,439.556,172.221,23.895,154.387
C01418=1067.606,-69.836,439.545,172.222,23.896,154.387
C01419=1067.613,-69.586,439.533,172.224,23.898,154.388
C01420=1067.618,-69.336,439.521,172.225,23.900,154.388
C01421=1067.624,-69.086,439.510,172.227,23.902,154.388
C01422=1067.630,-68.837,439.499,172.228,23.904,154.388
C01423=1067.637,-68.587,439.487,172.230,23.906,154.388
C01424=1067.643,-68.338,439.476,172.231,23.908,154.388
C01425=1067.648,-68.088,439.464,172.233,23.909,154.388
C01426=1067.654,-67.838,439.453,172.235,23.911,154.388
C01427=1067.661,-67.588,439.442,172.236,23.913,154.389
C01428=1067.667,-67.339,439.430,172.239,23.915,154.389
C01429=1067.672,-67.089,439.418,172.240,23.917,154.389
C01430=1067.678,-66.840,439.407,172.242,23.918,154.389
C01431=1067.685,-66.590,439.395,172.243,23.920,154.389
C01432=1067.691,-66.311,439.383,172.245,23.922,154.389
C01433=1067.698,-66.033,439.370,172.246,23.924,154.389
C01434=1067.705,-65.754,439.357,172.248,23.926,154.389
C01435=1067.711,-65.475,439.344,172.250,23.929,154.390
C01436=1067.717,-65.226,439.333,172.251,23.930,154.390
C01437=1067.724,-64.976,439.321,172.253,23.932,154.390
C01438=1067.730,-64.726,439.309,172.254,23.934,154.390
C01439=1067.735,-64.477,439.297,172.256,23.935,154.390
C01440=1067.742,-64.227,439.286,172.257,23.937,154.390
C01441=1067.748,-63.978,439.274,172.259,23.939,154.390
C01442=1067.754,-63.728,439.263,172.260,23.941,154.391
C01443=1067.759,-63.478,439.251,172.262,23.943,154.391
C01444=1067.766,-63.228,439.240,172.263,23.945,154.391
C01445=1067.772,-62.979,439.228,172.265,23.947,154.391
C01446=1067.777,-62.729,439.216,172.266,23.948,154.391
C01447=1067.784,-62.479,439.204,172.268,23.950,154.391
C01448=1067.790,-62.230,439.193,172.270,23.952,154.391
C01449=1067.796,-61.980,439.182,172.272,23.954,154.392
C01450=1067.802,-61.730,439.169,172.273,23.956,154.392
C01451=1067.808,-61.481,439.158,172.275,23.958,154.392
C01452=1067.815,-61.231,439.146,172.276,23.960,154.392
C01453=1067.821,-60.982,439.134,172.278,23.962,154.392
C01454=1067.826,-60.732,439.123,172.279,23.964,154.392
C01455=1067.833,-60.482,439.111,172.281,23.965,154.392
C01456=1067.839,-60.233,439.100,172.282,23.967,154.393
C01457=1067.844,-59.983,439.087,172.284,23.969,154.393
C01458=1067.851,-59.733,439.075,172.285,23.971,154.393
C01459=1067.857,-59.484,439.064,172.287,23.973,154.393
C01460=1067.863,-59.234,439.052,172.288,23.975,154.393
C01461=1067.869,-58.985,439.040,172.290,23.976,154.393
C01462=1067.875,-58.735,439.029,172.291,23.978,154.393
C01463=1067.881,-58.485,439.017,172.293,23.981,154.394
C01464=1067.888,-58.236,439.005,172.294,23.983,154.394
C01465=1067.893,-57.986,438.994,172.296,23.984,154.394
C01466=1067.900,-57.737,438.982,172.298,23.987,154.394
C01467=1067.906,-57.487,438.969,172.300,23.988,154.394
C01468=1067.912,-57.236,438.958,172.301,23.990,154.394
C01469=1067.918,-56.988,438.946,172.303,23.992,154.395
C01470=1067.924,-56.738,438.934,172.304,23.994,154.395
C01471=1067.931,-56.488,438.922,172.306,23.996,154.395
C01472=1067.936,-56.238,438.910,172.307,23.998,154.395
C01473=1067.943,-55.989,438.898,172.309,24.000,154.395
C01474=1067.949,-55.739,438.886,172.310,24.001,154.395
C01475=1067.955,-55.489,438.874,172.312,24.003,154.395
C01476=1067.961,-55.240,438.863,172.313,24.006,154.396
C01477=1067.968,-54.990,438.851,172.315,24.007,154.396
C01478=1067.973,-54.740,438.839,172.316,24.009,154.396
C01479=1067.980,-54.491,438.827,172.318,24.011,154.396
C01480=1067.986,-54.242,438.815,172.319,24.013,154.396
C01481=1067.992,-53.991,438.803,172.321,24.015,154.396
C01482=1067.998,-53.742,438.791,172.322,24.017,154.397
C01483=1068.005,-53.492,438.779,172.325,24.019,154.397
C01484=1068.010,-53.243,438.767,172.326,24.021,154.397
C01485=1068.017,-52.993,438.755,172.327,24.023,154.397
C01486=1068.023,-52.744,438.742,172.329,24.025,154.397
C01487=1068.029,-52.493,438.731,172.330,24.027,154.397
C01488=1068.036,-52.244,438.719,172.332,24.029,154.397
C01489=1068.041,-51.995,438.707,172.333,24.031,154.398
C01490=1068.048,-51.745,438.695,172.335,24.032,154.398
C01491=1068.054,-51.495,438.683,172.336,24.034,154.398
C01492=1068.060,-51.246,438.671,172.338,24.037,154.398
C01493=1068.067,-50.996,438.659,172.339,24.038,154.398
C01494=1068.072,-50.747,438.646,172.341,24.040,154.398
C01495=1068.079,-50.497,438.635,172.342,24.042,154.399
C01496=1068.086,-50.219,438.621,172.345,24.045,154.399
C01497=1068.093,-49.942,438.608,172.346,24.047,154.399
C01498=1068.099,-49.665,438.594,172.347,24.049,154.399
C01499=1068.106,-49.387,438.581,172.349,24.051,154.399
C01500=1068.111,-49.138,438.568,172.350,24.053,154.400
C01501=1068.118,-48.888,438.556,172.352,24.055,154.400
C01502=1068.123,-48.638,438.544,172.354,24.058,154.400
C01503=1068.129,-48.388,438.531,172.356,24.060,154.400
C01504=1068.135,-48.140,438.520,172.357,24.062,154.400
C01505=1068.141,-47.890,438.507,172.358,24.064,154.401
C01506=1068.147,-47.640,438.495,172.360,24.066,154.401
C01507=1068.154,-47.390,438.483,172.361,24.068,154.401
C01508=1068.160,-47.140,438.470,172.363,24.070,154.401
C01509=1068.165,-46.891,438.458,172.364,24.072,154.401
C01510=1068.172,-46.642,438.446,172.366,24.074,154.402
C01511=1068.178,-46.392,438.433,172.367,24.076,154.402
C01512=1068.184,-46.142,438.420,172.369,24.078,154.402
C01513=1068.190,-45.893,438.408,172.370,24.081,154.402
C01514=1068.196,-45.644,438.396,172.372,24.082,154.402
C01515=1068.202,-45.394,438.383,172.373,24.084,154.402
C01516=1068.208,-45.144,438.371,172.374,24.087,154.403
C01517=1068.214,-44.894,438.359,172.376,24.088,154.403
C01518=1068.220,-44.644,438.346,172.377,24.091,154.403
C01519=1068.226,-44.395,438.334,172.380,24.093,154.403
C01520=1068.231,-44.145,438.322,172.381,24.095,154.404
C01521=1068.238,-43.896,438.310,172.383,24.097,154.404
C01522=1068.244,-43.646,438.297,172.384,24.099,154.404
C01523=1068.250,-43.397,438.284,172.385,24.102,154.404
C01524=1068.257,-43.147,438.272,172.387,24.103,154.404
C01525=1068.263,-42.897,438.259,172.388,24.106,154.404
C01526=1068.269,-42.647,438.247,172.390,24.108,154.405
C01527=1068.274,-42.398,438.235,172.391,24.110,154.405
C01528=1068.281,-42.149,438.223,172.393,24.112,154.405
C01529=1068.287,-41.899,438.209,172.394,24.114,154.405
C01530=1068.293,-41.649,438.197,172.396,24.116,154.405
C01531=1068.299,-41.400,438.184,172.397,24.118,154.406
C01532=1068.305,-41.150,438.172,172.398,24.120,154.406
C01533=1068.311,-40.900,438.160,172.400,24.122,154.406
C01534=1068.317,-40.651,438.147,172.401,24.125,154.406
C01535=1068.323,-40.401,438.134,172.403,24.126,154.406
C01536=1068.330,-40.151,438.122,172.405,24.129,154.407
C01537=1068.335,-39.902,438.110,172.407,24.131,154.407
C01538=1068.341,-39.653,438.097,172.408,24.133,154.407
C01539=1068.347,-39.403,438.084,172.409,24.135,154.407
C01540=1068.353,-39.153,438.071,172.411,24.138,154.408
C01541=1068.360,-38.904,438.059,172.412,24.140,154.408
C01542=1068.366,-38.654,438.046,172.414,24.141,154.408
C01543=1068.372,-38.404,438.034,172.415,24.144,154.408
C01544=1068.378,-38.155,438.021,172.416,24.146,154.408
C01545=1068.384,-37.905,438.009,172.418,24.148,154.409
C01546=1068.390,-37.655,437.995,172.419,24.150,154.409
C01547=1068.396,-37.406,437.983,172.421,24.152,154.409
C01548=1068.402,-37.156,437.970,172.422,24.155,154.409
C01549=1068.407,-36.907,437.957,172.424,24.157,154.409
C01550=1068.413,-36.657,437.945,172.425,24.159,154.410
C01551=1068.419,-36.407,437.932,172.426,24.161,154.410
C01552=1068.425,-36.158,437.919,172.428,24.164,154.410
C01553=1068.431,-35.908,437.906,172.430,24.166,154.410
C01554=1068.437,-35.658,437.894,172.432,24.168,154.411
C01555=1068.444,-35.409,437.881,172.433,24.170,154.411
C01556=1068.449,-35.159,437.868,172.434,24.172,154.411
C01557=1068.456,-34.910,437.855,172.436,24.175,154.411
C01558=1068.462,-34.660,437.842,172.437,24.177,154.411
C01559=1068.467,-34.410,437.830,172.439,24.179,154.412
C01560=1068.474,-34.134,437.815,172.440,24.182,154.412
C01561=1068.480,-33.857,437.801,172.441,24.184,154.412
C01562=1068.488,-33.580,437.786,172.444,24.187,154.412
C01563=1068.494,-33.303,437.773,172.445,24.189,154.413
C01564=1068.500,-33.053,437.759,172.447,24.191,154.413
C01565=1068.506,-32.803,437.747,172.448,24.193,154.413
C01566=1068.512,-32.554,437.734,172.449,24.196,154.413
C01567=1068.518,-32.304,437.721,172.451,24.198,154.414
C01568=1068.524,-32.055,437.708,172.452,24.200,154.414
C01569=1068.530,-31.805,437.695,172.454,24.202,154.414
C01570=1068.537,-31.556,437.682,172.455,24.204,154.414
C01571=1068.542,-31.306,437.669,172.456,24.207,154.414
C01572=1068.549,-31.057,437.656,172.459,24.209,154.415
C01573=1068.555,-30.807,437.643,172.460,24.211,154.415
C01574=1068.561,-30.558,437.630,172.462,24.214,154.415
C01575=1068.567,-30.308,437.618,172.463,24.216,154.415
C01576=1068.573,-30.058,437.604,172.464,24.218,154.416
C01577=1068.579,-29.809,437.592,172.466,24.220,154.416
C01578=1068.585,-29.559,437.579,172.467,24.223,154.416
C01579=1068.591,-29.309,437.566,172.469,24.224,154.416
C01580=1068.598,-29.059,437.552,172.470,24.227,154.417
C01581=1068.604,-28.810,437.539,172.471,24.229,154.417
C01582=1068.610,-28.560,437.527,172.473,24.231,154.417
C01583=1068.616,-28.311,437.513,172.474,24.233,154.417
C01584=1068.622,-28.061,437.501,172.476,24.236,154.417
C01585=1068.628,-27.812,437.487,172.477,24.238,154.418
C01586=1068.634,-27.562,437.474,172.479,24.240,154.418
C01587=1068.640,-27.312,437.461,172.480,24.242,154.418
C01588=1068.646,-27.063,437.448,172.481,24.245,154.418
C01589=1068.652,-26.813,437.435,172.484,24.247,154.419
C01590=1068.658,-26.564,437.422,172.485,24.249,154.419
C01591=1068.664,-26.315,437.409,172.486,24.252,154.419
C01592=1068.669,-26.065,437.396,172.488,24.254,154.419
C01593=1068.676,-25.815,437.382,172.489,24.257,154.420
C01594=1068.682,-25.565,437.369,172.491,24.258,154.420
C01595=1068.688,-25.315,437.356,172.492,24.261,154.420
C01596=1068.694,-25.066,437.342,172.493,24.263,154.420
C01597=1068.700,-24.817,437.329,172.495,24.266,154.421
C01598=1068.706,-24.567,437.316,172.496,24.268,154.421
C01599=1068.712,-24.318,437.303,172.497,24.270,154.421
C01600=1068.718,-24.068,437.289,172.499,24.273,154.421
C01601=1068.724,-23.819,437.276,172.500,24.275,154.422
C01602=1068.730,-23.569,437.263,172.502,24.277,154.422
C01603=1068.735,-23.319,437.250,172.503,24.279,154.422
C01604=1068.741,-23.070,437.236,172.504,24.282,154.422
C01605=1068.748,-22.821,437.223,172.506,24.284,154.423
C01606=1068.754,-22.571,437.209,172.507,24.287,154.423
C01607=1068.760,-22.321,437.196,172.510,24.289,154.423
C01608=1068.766,-22.071,437.183,172.511,24.291,154.423
C01609=1068.772,-21.822,437.170,172.512,24.294,154.424
C01610=1068.777,-21.572,437.156,172.514,24.296,154.424
C01611=1068.784,-21.323,437.143,172.515,24.298,154.424
C01612=1068.790,-21.073,437.130,172.516,24.301,154.424
C01613=1068.795,-20.824,437.116,172.518,24.303,154.425
C01614=1068.802,-20.574,437.103,172.519,24.305,154.425
C01615=1068.808,-20.324,437.089,172.521,24.307,154.425
C01616=1068.814,-20.075,437.075,172.522,24.310,154.425
C01617=1068.820,-19.826,437.062,172.523,24.312,154.426
C01618=1068.826,-19.576,437.050,172.525,24.314,154.426
C01619=1068.831,-19.326,437.036,172.526,24.317,154.426
C01620=1068.838,-19.076,437.022,172.528,24.319,154.426
C01621=1068.844,-18.827,437.009,172.529,24.322,154.427
C01622=1068.850,-18.577,436.995,172.530,24.324,154.427
C01623=1068.856,-18.328,436.982,172.532,24.326,154.427
C01624=1068.862,-18.050,436.967,172.534,24.329,154.428
C01625=1068.870,-17.772,436.952,172.535,24.332,154.428
C01626=1068.876,-17.494,436.937,172.537,24.334,154.428
C01627=1068.883,-17.217,436.922,172.539,24.337,154.428
C01628=1068.889,-16.968,436.908,172.540,24.339,154.429
C01629=1068.895,-16.718,436.895,172.542,24.341,154.429
C01630=1068.901,-16.468,436.881,172.543,24.344,154.429
C01631=1068.907,-16.219,436.867,172.544,24.346,154.429
C01632=1068.913,-15.970,436.854,172.546,24.349,154.430
C01633=1068.919,-15.720,436.840,172.547,24.351,154.430
C01634=1068.926,-15.470,436.827,172.549,24.353,154.430
C01635=1068.932,-15.221,436.813,172.550,24.356,154.431
C01636=1068.937,-14.971,436.799,172.551,24.358,154.431
C01637=1068.944,-14.722,436.786,172.553,24.361,154.431
C01638=1068.950,-14.472,436.772,172.554,24.363,154.431
C01639=1068.956,-14.222,436.759,172.555,24.365,154.432
C01640=1068.961,-13.973,436.745,172.557,24.368,154.432
C01641=1068.967,-13.723,436.731,172.558,24.370,154.432
C01642=1068.973,-13.474,436.718,172.560,24.373,154.432
C01643=1068.979,-13.224,436.703,172.561,24.375,154.433
C01644=1068.985,-12.974,436.690,172.562,24.377,154.433
C01645=1068.991,-12.725,436.676,172.564,24.380,154.433
C01646=1068.997,-12.476,436.663,172.566,24.382,154.433
C01647=1069.003,-12.226,436.649,172.567,24.385,154.434
C01648=1069.009,-11.976,436.635,172.569,24.387,154.434
C01649=1069.015,-11.726,436.622,172.570,24.390,154.434
C01650=1069.021,-11.477,436.607,172.571,24.392,154.435
C01651=1069.027,-11.228,436.594,172.573,24.394,154.435
C01652=1069.033,-10.978,436.580,172.574,24.397,154.435
C01653=1069.038,-10.728,436.566,172.576,24.399,154.435
C01654=1069.045,-10.479,436.552,172.577,24.401,154.436
C01655=1069.051,-10.229,436.538,172.578,24.404,154.436
C01656=1069.057,-9.980,436.525,172.580,24.406,154.436
C01657=1069.063,-9.731,436.510,172.581,24.409,154.436
C01658=1069.068,-9.481,436.497,172.582,24.411,154.437
C01659=1069.075,-9.231,436.483,172.584,24.413,154.437
C01660=1069.080,-8.981,436.469,172.585,24.416,154.437
C01661=1069.087,-8.732,436.456,172.587,24.418,154.438
C01662=1069.093,-8.482,436.442,172.588,24.421,154.438
C01663=1069.099,-8.233,436.427,172.589,24.423,154.438
C01664=1069.105,-7.984,436.414,172.591,24.426,154.439
C01665=1069.111,-7.733,436.399,172.593,24.429,154.439
C01666=1069.117,-7.484,436.386,172.594,24.431,154.439
C01667=1069.123,-7.235,436.372,172.596,24.433,154.439
C01668=1069.129,-6.985,436.357,172.597,24.436,154.440
C01669=1069.135,-6.736,436.344,172.598,24.438,154.440
C01670=1069.141,-6.486,436.330,172.600,24.441,154.440
C01671=1069.147,-6.236,436.315,172.601,24.443,154.440
C01672=1069.153,-5.987,436.302,172.602,24.445,154.441
C01673=1069.159,-5.738,436.288,172.604,24.448,154.441
C01674=1069.165,-5.488,436.273,172.605,24.450,154.441
C01675=1069.171,-5.239,436.260,172.607,24.452,154.442
C01676=1069.177,-4.989,436.246,172.608,24.455,154.442
C01677=1069.183,-4.739,436.232,172.609,24.457,154.442
C01678=1069.189,-4.490,436.218,172.611,24.460,154.442
C01679=1069.195,-4.240,436.204,172.612,24.463,154.443
C01680=1069.201,-3.990,436.190,172.613,24.465,154.443
C01681=1069.207,-3.742,436.176,172.615,24.467,154.443
C01682=1069.213,-3.491,436.162,172.616,24.470,154.444
C01683=1069.219,-3.242,436.148,172.617,24.472,154.444
C01684=1069.225,-2.993,436.134,172.619,24.474,154.444
C01685=1069.232,-2.743,436.119,172.621,24.477,154.444
C01686=1069.237,-2.494,436.105,172.622,24.480,154.445
C01687=1069.243,-2.244,436.091,172.624,24.482,154.445
C01688=1069.249,-1.965,436.075,172.625,24.485,154.445
C01689=1069.256,-1.685,436.059,172.626,24.488,154.446
C01690=1069.262,-1.406,436.043,172.628,24.491,154.446
C01691=1069.270,-1.127,436.027,172.630,24.493,154.446
C01692=1069.275,-0.877,436.013,172.631,24.496,154.447
C01693=1069.281,-0.627,435.999,172.633,24.499,154.447
C01694=1069.287,-0.378,435.984,172.634,24.501,154.447
C01695=1069.293,-0.129,435.970,172.635,24.504,154.448
C01696=1069.299,0.121,435.955,172.637,24.506,154.448
C01697=1069.304,0.371,435.942,172.638,24.509,154.448
C01698=1069.310,0.620,435.927,172.639,24.511,154.449
C01699=1069.316,0.870,435.913,172.641,24.514,154.449
C01700=1069.322,1.119,435.898,172.642,24.516,154.449
C01701=1069.328,1.369,435.884,172.643,24.519,154.449
C01702=1069.334,1.618,435.869,172.645,24.521,154.450
C01703=1069.339,1.868,435.856,172.646,24.524,154.450
C01704=1069.346,2.117,435.841,172.647,24.526,154.450
C01705=1069.351,2.367,435.827,172.649,24.529,154.451
C01706=1069.358,2.617,435.812,172.650,24.531,154.451
C01707=1069.363,2.865,435.797,172.652,24.534,154.451
C01708=1069.370,3.115,435.784,172.654,24.536,154.451
C01709=1069.376,3.364,435.769,172.655,24.539,154.452
C01710=1069.382,3.614,435.755,172.656,24.542,154.452
C01711=1069.388,3.864,435.740,172.658,24.544,154.452
C01712=1069.393,4.113,435.726,172.659,24.546,154.453
C01713=1069.400,4.363,435.711,172.661,24.549,154.453
C01714=1069.406,4.612,435.697,172.662,24.552,154.453
C01715=1069.412,4.862,435.683,172.663,24.554,154.454
C01716=1069.417,5.111,435.668,172.665,24.557,154.454
C01717=1069.424,5.361,435.653,172.666,24.559,154.454
C01718=1069.429,5.610,435.639,172.667,24.562,154.455
C01719=1069.436,5.860,435.624,172.669,24.564,154.455
C01720=1069.441,6.109,435.610,172.670,24.567,154.455
C01721=1069.448,6.359,435.595,172.671,24.569,154.455
C01722=1069.453,6.608,435.581,172.673,24.572,154.456
C01723=1069.460,6.858,435.566,172.674,24.574,154.456
C01724=1069.465,7.107,435.552,172.675,24.577,154.456
C01725=1069.472,7.357,435.537,172.677,24.579,154.457
C01726=1069.477,7.606,435.522,172.678,24.582,154.457
C01727=1069.483,7.856,435.508,172.679,24.584,154.457
C01728=1069.489,8.105,435.494,172.681,24.587,154.458
C01729=1069.496,8.355,435.479,172.683,24.589,154.458
C01730=1069.501,8.604,435.464,172.684,24.592,154.458
C01731=1069.507,8.854,435.450,172.686,24.595,154.459
C01732=1069.513,9.103,435.435,172.687,24.597,154.459
C01733=1069.520,9.353,435.420,172.688,24.599,154.459
C01734=1069.525,9.602,435.405,172.690,24.602,154.459
C01735=1069.531,9.852,435.391,172.691,24.605,154.460
C01736=1069.537,10.102,435.376,172.692,24.607,154.460
C01737=1069.543,10.351,435.361,172.694,24.610,154.460
C01738=1069.549,10.601,435.347,172.695,24.612,154.461
C01739=1069.555,10.850,435.333,172.696,24.615,154.461
C01740=1069.561,11.100,435.318,172.698,24.617,154.461
C01741=1069.567,11.349,435.303,172.699,24.620,154.462
C01742=1069.573,11.598,435.288,172.700,24.622,154.462
C01743=1069.580,11.848,435.273,172.702,24.625,154.462
C01744=1069.585,12.097,435.259,172.703,24.627,154.463
C01745=1069.592,12.347,435.244,172.705,24.630,154.463
C01746=1069.597,12.596,435.230,172.706,24.633,154.463
C01747=1069.604,12.846,435.215,172.707,24.635,154.463
C01748=1069.610,13.096,435.200,172.709,24.637,154.464
C01749=1069.616,13.344,435.185,172.710,24.640,154.464
C01750=1069.622,13.594,435.170,172.711,24.643,154.464
C01751=1069.628,13.844,435.155,172.714,24.645,154.465
C01752=1069.635,14.125,435.139,172.715,24.648,154.465
C01753=1069.641,14.406,435.122,172.716,24.651,154.465
C01754=1069.648,14.688,435.105,172.718,24.654,154.466
C01755=1069.655,14.969,435.088,172.720,24.657,154.466
C01756=1069.661,15.219,435.073,172.721,24.659,154.466
C01757=1069.667,15.468,435.059,172.722,24.662,154.467
C01758=1069.673,15.717,435.044,172.724,24.664,154.467
C01759=1069.679,15.967,435.028,172.725,24.667,154.467
C01760=1069.685,16.216,435.014,172.726,24.670,154.468
C01761=1069.691,16.466,434.999,172.728,24.672,154.468
C01762=1069.696,16.715,434.984,172.729,24.674,154.468
C01763=1069.702,16.965,434.969,172.730,24.677,154.469
C01764=1069.709,17.214,434.954,172.732,24.680,154.469
C01765=1069.715,17.463,434.939,172.733,24.682,154.469
C01766=1069.720,17.713,434.924,172.734,24.685,154.470
C01767=1069.727,17.963,434.909,172.736,24.687,154.470
C01768=1069.732,18.212,434.894,172.737,24.690,154.470
C01769=1069.738,18.462,434.879,172.738,24.693,154.471
C01770=1069.744,18.712,434.864,172.740,24.695,154.471
C01771=1069.750,18.960,434.849,172.741,24.697,154.471
C01772=1069.756,19.210,434.833,172.743,24.701,154.471
C01773=1069.762,19.460,434.819,172.745,24.703,154.472
C01774=1069.768,19.709,434.804,172.746,24.706,154.472
C01775=1069.774,19.959,434.788,172.747,24.708,154.472
C01776=1069.780,20.209,434.773,172.749,24.711,154.473
C01777=1069.786,20.458,434.759,172.750,24.714,154.473
C01778=1069.791,20.708,434.743,172.752,24.716,154.473
C01779=1069.798,20.957,434.728,172.753,24.718,154.474
C01780=1069.803,21.206,434.713,172.754,24.721,154.474
C01781=1069.810,21.456,434.698,172.756,24.724,154.474
C01782=1069.816,21.705,434.683,172.757,24.727,154.475
C01783=1069.821,21.955,434.667,172.758,24.729,154.475
C01784=1069.827,22.204,434.653,172.759,24.732,154.475
C01785=1069.833,22.454,434.637,172.761,24.734,154.476
C01786=1069.839,22.702,434.622,172.762,24.737,154.476
C01787=1069.845,22.952,434.606,172.764,24.740,154.476
C01788=1069.851,23.202,434.591,172.765,24.742,154.477
C01789=1069.857,23.451,434.577,172.766,24.745,154.477
C01790=1069.863,23.701,434.561,172.768,24.747,154.477
C01791=1069.869,23.950,434.545,172.769,24.750,154.478
C01792=1069.875,24.200,434.530,172.770,24.752,154.478
C01793=1069.881,24.449,434.515,172.773,24.755,154.478
C01794=1069.886,24.699,434.500,172.774,24.758,154.479
C01795=1069.893,24.948,434.484,172.775,24.760,154.479
C01796=1069.898,25.197,434.469,172.777,24.763,154.479
C01797=1069.904,25.447,434.454,172.778,24.766,154.480
C01798=1069.910,25.697,434.438,172.779,24.768,154.480
C01799=1069.917,25.946,434.423,172.781,24.771,154.480
C01800=1069.922,26.195,434.408,172.782,24.773,154.481
C01801=1069.928,26.445,434.393,172.783,24.776,154.481
C01802=1069.934,26.695,434.377,172.785,24.779,154.481
C01803=1069.941,26.944,434.361,172.786,24.781,154.482
C01804=1069.946,27.194,434.346,172.787,24.784,154.482
C01805=1069.952,27.443,434.331,172.789,24.786,154.482
C01806=1069.958,27.692,434.315,172.790,24.789,154.483
C01807=1069.964,27.942,434.300,172.791,24.792,154.483
C01808=1069.970,28.192,434.285,172.793,24.794,154.483
C01809=1069.976,28.440,434.269,172.794,24.797,154.484
C01810=1069.982,28.690,434.254,172.795,24.799,154.484
C01811=1069.988,28.939,434.238,172.797,24.802,154.484
C01812=1069.994,29.189,434.223,172.798,24.804,154.485
C01813=1069.999,29.438,434.207,172.800,24.808,154.485
C01814=1070.006,29.687,434.192,172.802,24.810,154.485
C01815=1070.011,29.937,434.176,172.803,24.813,154.486
C01816=1070.018,30.220,434.158,172.804,24.816,154.486
C01817=1070.024,30.502,434.140,172.805,24.819,154.486
